	LOCAL CONST Robtarget Tr_meulage_bavure_P270 :=[[-219.63696875,-205.171546875,20],[0.53729501780428,-0.564922938891818,0.453775369108491,-0.431583191687283],[0,0,0,0],[8.999999E+09,8.999999E+09,8.999999E+09,8.999999E+09,8.999999E+09,8.999999E+09]];
	LOCAL CONST Robtarget Tr_meulage_bavure_P271 :=[[-219.324734375,-207.44634375,20],[0.537993238973984,-0.564758927457813,0.45310570554085,-0.431631611772482],[0,0,0,0],[8.999999E+09,8.999999E+09,8.999999E+09,8.999999E+09,8.999999E+09,8.999999E+09]];
	LOCAL CONST Robtarget Tr_meulage_bavure_P272 :=[[-219.077484375,-208.372515625,20],[0.538304707849301,-0.564135132378618,0.452955772497051,-0.432215990084863],[0,0,0,0],[8.999999E+09,8.999999E+09,8.999999E+09,8.999999E+09,8.999999E+09,8.999999E+09]];
	LOCAL CONST Robtarget Tr_meulage_bavure_P273 :=[[-218.728875,-210.97625,20],[0.538253392960368,-0.56310894895446,0.453282288328033,-0.433274466893857],[0,0,0,0],[8.999999E+09,8.999999E+09,8.999999E+09,8.999999E+09,8.999999E+09,8.999999E+09]];
	LOCAL CONST Robtarget Tr_meulage_bavure_P274 :=[[-218.566671875,-211.56171875,20],[0.537902797214692,-0.561749600415359,0.453996649502375,-0.434724061241626],[0,0,0,0],[8.999999E+09,8.999999E+09,8.999999E+09,8.999999E+09,8.999999E+09,8.999999E+09]];
	LOCAL CONST Robtarget Tr_meulage_bavure_P275 :=[[-217.610703125,-218.654484375,20],[0.537331594068803,-0.560152131881694,0.454988034586502,-0.436451870825392],[0,0,0,0],[8.999999E+09,8.999999E+09,8.999999E+09,8.999999E+09,8.999999E+09,8.999999E+09]];
	LOCAL CONST Robtarget Tr_meulage_bavure_P276 :=[[-217.24321875,-220.540375,20],[0.536643862605788,-0.558402103153409,0.456123837189228,-0.438350888067042],[0,0,0,0],[8.999999E+09,8.999999E+09,8.999999E+09,8.999999E+09,8.999999E+09,8.999999E+09]];
	LOCAL CONST Robtarget Tr_meulage_bavure_P277 :=[[-217.107078125,-221.269171875,20],[0.535921621847869,-0.55659175325912,0.457294923702402,-0.440312375701505],[0,0,0,0],[8.999999E+09,8.999999E+09,8.999999E+09,8.999999E+09,8.999999E+09,8.999999E+09]];
	LOCAL CONST Robtarget Tr_meulage_bavure_P278 :=[[-216.99709375,-221.83040625,20],[0.535229940524766,-0.55481109003148,0.458413067683216,-0.44223412862555],[0,0,0,0],[8.999999E+09,8.999999E+09,8.999999E+09,8.999999E+09,8.999999E+09,8.999999E+09]];
	LOCAL CONST Robtarget Tr_meulage_bavure_P279 :=[[-215.919453125,-225.61296875,20],[0.534637158213425,-0.553121918752511,0.459395983531932,-0.44404344648665],[0,0,0,0],[8.999999E+09,8.999999E+09,8.999999E+09,8.999999E+09,8.999999E+09,8.999999E+09]];
	LOCAL CONST Robtarget Tr_meulage_bavure_P280 :=[[-215.4938125,-227.822453125,20],[0.534190972566451,-0.551569737548126,0.460187785384334,-0.445688267326685],[0,0,0,0],[8.999999E+09,8.999999E+09,8.999999E+09,8.999999E+09,8.999999E+09,8.999999E+09]];
	LOCAL CONST Robtarget Tr_meulage_bavure_P281 :=[[-215.101453125,-230.017,20],[0.533919682326157,-0.550203109380352,0.460752711338939,-0.447116595807787],[0,0,0,0],[8.999999E+09,8.999999E+09,8.999999E+09,8.999999E+09,8.999999E+09,8.999999E+09]];
	LOCAL CONST Robtarget Tr_meulage_bavure_P282 :=[[-214.766375,-231.03446875,20],[0.533869793524164,-0.549045269612884,0.461042387233755,-0.448299289149539],[0,0,0,0],[8.999999E+09,8.999999E+09,8.999999E+09,8.999999E+09,8.999999E+09,8.999999E+09]];
	LOCAL CONST Robtarget Tr_meulage_bavure_P283 :=[[-214.39034375,-233.601546875,20],[0.534074564116095,-0.548144938680638,0.461016631292879,-0.449182759947851],[0,0,0,0],[8.999999E+09,8.999999E+09,8.999999E+09,8.999999E+09,8.999999E+09,8.999999E+09]];
	LOCAL CONST Robtarget Tr_meulage_bavure_P284 :=[[-214.230546875,-234.2085625,20],[0.534566009335567,-0.547535508259174,0.460639359023246,-0.449728173208069],[0,0,0,0],[8.999999E+09,8.999999E+09,8.999999E+09,8.999999E+09,8.999999E+09,8.999999E+09]];
	LOCAL CONST Robtarget Tr_meulage_bavure_P285 :=[[-213.2238125,-241.16003125,20],[0.535386335741234,-0.547259939100456,0.459861332170375,-0.449883969187421],[0,0,0,0],[8.999999E+09,8.999999E+09,8.999999E+09,8.999999E+09,8.999999E+09,8.999999E+09]];
	LOCAL CONST Robtarget Tr_meulage_bavure_P286 :=[[-212.793484375,-243.30528125,20],[0.536594038742582,-0.547390070776213,0.458609537333498,-0.449564500676256],[0,0,0,0],[8.999999E+09,8.999999E+09,8.999999E+09,8.999999E+09,8.999999E+09,8.999999E+09]];
	LOCAL CONST Robtarget Tr_meulage_bavure_P287 :=[[-212.653484375,-243.93984375,20],[0.538255330930929,-0.54797778261946,0.456804384011849,-0.448699569007427],[0,0,0,0],[8.999999E+09,8.999999E+09,8.999999E+09,8.999999E+09,8.999999E+09,8.999999E+09]];
	LOCAL CONST Robtarget Tr_meulage_bavure_P288 :=[[-212.53553125,-244.61078125,20],[0.540450412619775,-0.549105109829106,0.454341727655778,-0.447180639528864],[0,0,0,0],[8.999999E+09,8.999999E+09,8.999999E+09,8.999999E+09,8.999999E+09,8.999999E+09]];
	LOCAL CONST Robtarget Tr_meulage_bavure_P289 :=[[-211.432546875,-248.382609375,20],[0.543265483790806,-0.550855839481898,0.451104099741733,-0.44488824374941],[0,0,0,0],[8.999999E+09,8.999999E+09,8.999999E+09,8.999999E+09,8.999999E+09,8.999999E+09]];
	LOCAL CONST Robtarget Tr_meulage_bavure_P290 :=[[-210.87403125,-250.098296875,20],[0.546796245142534,-0.553313577146664,0.446954285400637,-0.441689730925675],[0,0,0,0],[8.999999E+09,8.999999E+09,8.999999E+09,8.999999E+09,8.999999E+09,8.999999E+09]];
	LOCAL CONST Robtarget Tr_meulage_bavure_P291 :=[[-210.5504375,-252.859703125,20],[0.551129613263795,-0.556588605739961,0.441743303392717,-0.43741070774712],[0,0,0,0],[8.999999E+09,8.999999E+09,8.999999E+09,8.999999E+09,8.999999E+09,8.999999E+09]];
	LOCAL CONST Robtarget Tr_meulage_bavure_P292 :=[[-210.326328125,-253.7085625,20],[0.556352636409364,-0.560749575377414,0.435311239016695,-0.431897884759985],[0,0,0,0],[8.999999E+09,8.999999E+09,8.999999E+09,8.999999E+09,8.999999E+09,8.999999E+09]];
	LOCAL CONST Robtarget Tr_meulage_bavure_P293 :=[[-209.778859375,-256.37915625,20],[0.562534887167558,-0.565860689136051,0.427491552289097,-0.424979004106455],[0,0,0,0],[8.999999E+09,8.999999E+09,8.999999E+09,8.999999E+09,8.999999E+09,8.999999E+09]];
	LOCAL CONST Robtarget Tr_meulage_bavure_P294 :=[[-209.6011875,-256.862328125,20],[0.569700795502199,-0.571957017682978,0.418140443553853,-0.416490987888025],[0,0,0,0],[8.999999E+09,8.999999E+09,8.999999E+09,8.999999E+09,8.999999E+09,8.999999E+09]];
	LOCAL CONST Robtarget Tr_meulage_bavure_P295 :=[[-208.96625,-259.827125,20],[0.577848420825114,-0.579022623980751,0.407121335426489,-0.406295731836946],[0,0,0,0],[8.999999E+09,8.999999E+09,8.999999E+09,8.999999E+09,8.999999E+09,8.999999E+09]];
	LOCAL CONST Robtarget Tr_meulage_bavure_P296 :=[[-208.80403125,-260.40115625,20],[0.586930696044148,-0.586995327394604,0.394324157697137,-0.394280740481293],[0,0,0,0],[8.999999E+09,8.999999E+09,8.999999E+09,8.999999E+09,8.999999E+09,8.999999E+09]];
	LOCAL CONST Robtarget Tr_meulage_bavure_P297 :=[[-206.9465625,-264.3128125,20],[0.596830556528174,-0.595758661219479,0.379700963340443,-0.380384125345135],[0,0,0,0],[8.999999E+09,8.999999E+09,8.999999E+09,8.999999E+09,8.999999E+09,8.999999E+09]];
	LOCAL CONST Robtarget Tr_meulage_bavure_P298 :=[[-204.21284375,-269.3765625,20],[0.607373754979424,-0.60515091678245,0.363261810220388,-0.364596142210751],[0,0,0,0],[8.999999E+09,8.999999E+09,8.999999E+09,8.999999E+09,8.999999E+09,8.999999E+09]];
	LOCAL CONST Robtarget Tr_meulage_bavure_P299 :=[[-204.11028125,-269.53403125,20],[0.618359765363299,-0.61496081647422,0.345061273014783,-0.346968460593501],[0,0,0,0],[8.999999E+09,8.999999E+09,8.999999E+09,8.999999E+09,8.999999E+09,8.999999E+09]];
	LOCAL CONST Robtarget Tr_meulage_bavure_P300 :=[[-203.988234375,-269.722875,20],[0.629554145495922,-0.624946065590333,0.325221808959532,-0.327619852831222],[0,0,0,0],[8.999999E+09,8.999999E+09,8.999999E+09,8.999999E+09,8.999999E+09,8.999999E+09]];
	LOCAL CONST Robtarget Tr_meulage_bavure_P301 :=[[-202.10503125,-271.81009375,20],[0.640691980291868,-0.634846776112635,0.303952512068475,-0.306751084197502],[0,0,0,0],[8.999999E+09,8.999999E+09,8.999999E+09,8.999999E+09,8.999999E+09,8.999999E+09]];
	LOCAL CONST Robtarget Tr_meulage_bavure_P302 :=[[-198.574953125,-275.987625,20],[0.651514894985457,-0.64441431008127,0.28151592453752,-0.284617853983822],[0,0,0,0],[8.999999E+09,8.999999E+09,8.999999E+09,8.999999E+09,8.999999E+09,8.999999E+09]];
	LOCAL CONST Robtarget Tr_meulage_bavure_P303 :=[[-198.1525625,-276.32359375,20],[0.661778551172858,-0.653403298900412,0.258256180431549,-0.261566480005598],[0,0,0,0],[8.999999E+09,8.999999E+09,8.999999E+09,8.999999E+09,8.999999E+09,8.999999E+09]];
	LOCAL CONST Robtarget Tr_meulage_bavure_P304 :=[[-198.02296875,-276.43640625,20],[0.671270334947485,-0.661609679683465,0.234574203209948,-0.237999395707325],[0,0,0,0],[8.999999E+09,8.999999E+09,8.999999E+09,8.999999E+09,8.999999E+09,8.999999E+09]];
	LOCAL CONST Robtarget Tr_meulage_bavure_P305 :=[[-193.361921875,-279.8115,20],[0.679821587865466,-0.668886501373737,0.210911256713211,-0.214359274918843],[0,0,0,0],[8.999999E+09,8.999999E+09,8.999999E+09,8.999999E+09,8.999999E+09,8.999999E+09]];
	LOCAL CONST Robtarget Tr_meulage_bavure_P306 :=[[-192.662015625,-280.25846875,20],[0.687332808397279,-0.675135741510664,0.187723907861307,-0.191115345937563],[0,0,0,0],[8.999999E+09,8.999999E+09,8.999999E+09,8.999999E+09,8.999999E+09,8.999999E+09]];
	LOCAL CONST Robtarget Tr_meulage_bavure_P307 :=[[-185.646046875,-284.1375,20],[0.693782149187908,-0.680318577808721,0.165437229325596,-0.168711248319718],[0,0,0,0],[8.999999E+09,8.999999E+09,8.999999E+09,8.999999E+09,8.999999E+09,8.999999E+09]];
	LOCAL CONST Robtarget Tr_meulage_bavure_P308 :=[[-185.354671875,-284.25996875,20],[0.699188719439392,-0.684470610463102,0.144444095505406,-0.147550063688893],[0,0,0,0],[8.999999E+09,8.999999E+09,8.999999E+09,8.999999E+09,8.999999E+09,8.999999E+09]];
	LOCAL CONST Robtarget Tr_meulage_bavure_P309 :=[[-180.695234375,-286.03475,20],[0.70362823463154,-0.687682408745583,0.125033593354582,-0.127932844352095],[0,0,0,0],[8.999999E+09,8.999999E+09,8.999999E+09,8.999999E+09,8.999999E+09,8.999999E+09]];
	LOCAL CONST Robtarget Tr_meulage_bavure_P310 :=[[-179.823375,-286.31721875,20],[0.707229971052489,-0.690061561664037,0.107377724376658,-0.110049232012663],[0,0,0,0],[8.999999E+09,8.999999E+09,8.999999E+09,8.999999E+09,8.999999E+09,8.999999E+09]];
	LOCAL CONST Robtarget Tr_meulage_bavure_P311 :=[[-179.685515625,-286.362125,20],[0.71011625284017,-0.691753966347935,0.0915438463828495,-0.0939738351008869],[0,0,0,0],[8.999999E+09,8.999999E+09,8.999999E+09,8.999999E+09,8.999999E+09,8.999999E+09]];
	LOCAL CONST Robtarget Tr_meulage_bavure_P312 :=[[-179.47846875,-286.4050625,20],[0.712422501657508,-0.692893522682186,0.0774902952212525,-0.0796743340333189],[0,0,0,0],[8.999999E+09,8.999999E+09,8.999999E+09,8.999999E+09,8.999999E+09,8.999999E+09]];
	LOCAL CONST Robtarget Tr_meulage_bavure_P313 :=[[-176.450546875,-286.82434375,20],[0.714278213115217,-0.693598764499872,0.0650809529079148,-0.0670213228889187],[0,0,0,0],[8.999999E+09,8.999999E+09,8.999999E+09,8.999999E+09,8.999999E+09,8.999999E+09]];
	LOCAL CONST Robtarget Tr_meulage_bavure_P314 :=[[-174.725015625,-287.0270625,20],[0.715791157369704,-0.693969981495662,0.0541362999646006,-0.0558385605150519],[0,0,0,0],[8.999999E+09,8.999999E+09,8.999999E+09,8.999999E+09,8.999999E+09,8.999999E+09]];
	LOCAL CONST Robtarget Tr_meulage_bavure_P315 :=[[-172.48009375,-287.12125,20],[0.717041268538116,-0.694095069222552,0.0444470233568255,-0.045916404572963],[0,0,0,0],[8.999999E+09,8.999999E+09,8.999999E+09,8.999999E+09,8.999999E+09,8.999999E+09]];
	LOCAL CONST Robtarget Tr_meulage_bavure_P316 :=[[-170.3138125,-287.373625,20],[0.718086151112885,-0.694044263785635,0.0358082882651692,-0.0370486973813791],[0,0,0,0],[8.999999E+09,8.999999E+09,8.999999E+09,8.999999E+09,8.999999E+09,8.999999E+09]];
	LOCAL CONST Robtarget Tr_meulage_bavure_P317 :=[[-169.579875,-287.35590625,20],[0.718985888631994,-0.693850501788261,0.0280425230376692,-0.0290583898026416],[0,0,0,0],[8.999999E+09,8.999999E+09,8.999999E+09,8.999999E+09,8.999999E+09,8.999999E+09]];
	LOCAL CONST Robtarget Tr_meulage_bavure_P318 :=[[-166.023984375,-287.1190625,20],[0.719774919648292,-0.693547646838508,0.0209970440043696,-0.0217910704909592],[0,0,0,0],[8.999999E+09,8.999999E+09,8.999999E+09,8.999999E+09,8.999999E+09,8.999999E+09]];
	LOCAL CONST Robtarget Tr_meulage_bavure_P319 :=[[-160.928265625,-287.3099375,20],[0.720464951309386,-0.693172347648877,0.0145821147957829,-0.0151562633188785],[0,0,0,0],[8.999999E+09,8.999999E+09,8.999999E+09,8.999999E+09,8.999999E+09,8.999999E+09]];
	LOCAL CONST Robtarget Tr_meulage_bavure_P320 :=[[-160.79965625,-287.30678125,20],[0.721085760434946,-0.692731207117006,0.00873022747837951,-0.00908756911099294],[0,0,0,0],[8.999999E+09,8.999999E+09,8.999999E+09,8.999999E+09,8.999999E+09,8.999999E+09]];
	LOCAL CONST Robtarget Tr_meulage_bavure_P321 :=[[-158.17290625,-287.03840625,20],[0.721652690962883,-0.692237672883823,0.00341929407178484,-0.00356458896236797],[0,0,0,0],[8.999999E+09,8.999999E+09,8.999999E+09,8.999999E+09,8.999999E+09,8.999999E+09]];
	LOCAL CONST Robtarget Tr_meulage_bavure_P322 :=[[-156.189484375,-287.00271875,20],[0.722168553326168,-0.691714363171503,-0.00135201117505688,0.00141153633111643],[0,0,0,0],[8.999999E+09,8.999999E+09,8.999999E+09,8.999999E+09,8.999999E+09,8.999999E+09]];
	LOCAL CONST Robtarget Tr_meulage_bavure_P323 :=[[-152.667203125,-287.19778125,20],[0.722648884556597,-0.691168089401874,-0.00558376990281725,0.00583809518084595],[0,0,0,0],[8.999999E+09,8.999999E+09,8.999999E+09,8.999999E+09,8.999999E+09,8.999999E+09]];
	LOCAL CONST Robtarget Tr_meulage_bavure_P324 :=[[-149.589046875,-287.21059375,20],[0.723113666831497,-0.690599316019845,-0.00924582442862393,0.00968113036079282],[0,0,0,0],[8.999999E+09,8.999999E+09,8.999999E+09,8.999999E+09,8.999999E+09,8.999999E+09]];
	LOCAL CONST Robtarget Tr_meulage_bavure_P325 :=[[-144.85625,-286.99990625,20],[0.72355718246237,-0.690033503818427,-0.0123218608697659,0.0129204899244532],[0,0,0,0],[8.999999E+09,8.999999E+09,8.999999E+09,8.999999E+09,8.999999E+09,8.999999E+09]];
	LOCAL CONST Robtarget Tr_meulage_bavure_P326 :=[[-143.57653125,-287.2320625,20],[0.723999358467151,-0.689466631061457,-0.0148019658892337,0.0155433393366104],[0,0,0,0],[8.999999E+09,8.999999E+09,8.999999E+09,8.999999E+09,8.999999E+09,8.999999E+09]];
	LOCAL CONST Robtarget Tr_meulage_bavure_P327 :=[[-140.72509375,-287.0025,20],[0.724444298776135,-0.688908293410537,-0.0166790464051948,0.0175394028390153],[0,0,0,0],[8.999999E+09,8.999999E+09,8.999999E+09,8.999999E+09,8.999999E+09,8.999999E+09]];
	LOCAL CONST Robtarget Tr_meulage_bavure_P328 :=[[-139.5401875,-286.91978125,20],[0.72490078853614,-0.688359587713625,-0.0179553342944921,0.0189084836193525],[0,0,0,0],[8.999999E+09,8.999999E+09,8.999999E+09,8.999999E+09,8.999999E+09,8.999999E+09]];
	LOCAL CONST Robtarget Tr_meulage_bavure_P329 :=[[-137.21515625,-287.07465625,20],[0.725359692131602,-0.687835653160883,-0.0186601652392554,0.0196781478989506],[0,0,0,0],[8.999999E+09,8.999999E+09,8.999999E+09,8.999999E+09,8.999999E+09,8.999999E+09]];
	LOCAL CONST Robtarget Tr_meulage_bavure_P330 :=[[-135.483828125,-287.07825,20],[0.725833732047821,-0.687323758836874,-0.0188483306036036,0.0199043812599118],[0,0,0,0],[8.999999E+09,8.999999E+09,8.999999E+09,8.999999E+09,8.999999E+09,8.999999E+09]];
	LOCAL CONST Robtarget Tr_meulage_bavure_P331 :=[[-132.387421875,-286.80325,20],[0.726321044579261,-0.686822734580372,-0.018592585476214,0.0196618216383935],[0,0,0,0],[8.999999E+09,8.999999E+09,8.999999E+09,8.999999E+09,8.999999E+09,8.999999E+09]];
	LOCAL CONST Robtarget Tr_meulage_bavure_P332 :=[[-130.4786953125,-286.93715625,20],[0.726812176110579,-0.68633672027097,-0.0179819950748647,0.0190424504258088],[0,0,0,0],[8.999999E+09,8.999999E+09,8.999999E+09,8.999999E+09,8.999999E+09,8.999999E+09]];
	LOCAL CONST Robtarget Tr_meulage_bavure_P333 :=[[-129.3878515625,-286.88765625,20],[0.727297328990863,-0.685868930510056,-0.0171164226950637,0.0181503024181905],[0,0,0,0],[8.999999E+09,8.999999E+09,8.999999E+09,8.999999E+09,8.999999E+09,8.999999E+09]];
	LOCAL CONST Robtarget Tr_meulage_bavure_P334 :=[[-126.4455859375,-287.0436875,20],[0.727787757509097,-0.68540016068255,-0.0161018599931864,0.0170976565930428],[0,0,0,0],[8.999999E+09,8.999999E+09,8.999999E+09,8.999999E+09,8.999999E+09,8.999999E+09]];
	LOCAL CONST Robtarget Tr_meulage_bavure_P335 :=[[-126.3676171875,-287.04559375,20],[0.72827628013861,-0.684932120707197,-0.0150354989508349,0.0159869816510227],[0,0,0,0],[8.999999E+09,8.999999E+09,8.999999E+09,8.999999E+09,8.999999E+09,8.999999E+09]];
	LOCAL CONST Robtarget Tr_meulage_bavure_P336 :=[[-122.262265625,-286.86140625,20],[0.728755053664664,-0.684469256132264,-0.0139954111703684,0.0149009272909549],[0,0,0,0],[8.999999E+09,8.999999E+09,8.999999E+09,8.999999E+09,8.999999E+09,8.999999E+09]];
	LOCAL CONST Robtarget Tr_meulage_bavure_P337 :=[[-120.081265625,-287.044,20],[0.729234909118417,-0.683998119330656,-0.0130346409279294,0.0138966978473149],[0,0,0,0],[8.999999E+09,8.999999E+09,8.999999E+09,8.999999E+09,8.999999E+09,8.999999E+09]];
	LOCAL CONST Robtarget Tr_meulage_bavure_P338 :=[[-118.7465546875,-287.03021875,20],[0.729708993844251,-0.683525414703059,-0.0121869491838472,0.013010381524496],[0,0,0,0],[8.999999E+09,8.999999E+09,8.999999E+09,8.999999E+09,8.999999E+09,8.999999E+09]];
	LOCAL CONST Robtarget Tr_meulage_bavure_P339 :=[[-116.7078515625,-287.04834375,20],[0.730167601402134,-0.683061652581515,-0.011473244296343,0.0122644731064913],[0,0,0,0],[8.999999E+09,8.999999E+09,8.999999E+09,8.999999E+09,8.999999E+09,8.999999E+09]];
	LOCAL CONST Robtarget Tr_meulage_bavure_P340 :=[[-116.34390625,-287.02965625,20],[0.730618690391253,-0.682598813248682,-0.0109056678682374,0.0116728664349885],[0,0,0,0],[8.999999E+09,8.999999E+09,8.999999E+09,8.999999E+09,8.999999E+09,8.999999E+09]];
	LOCAL CONST Robtarget Tr_meulage_bavure_P341 :=[[-115.980984375,-287.02528125,20],[0.731069622640329,-0.682129611176638,-0.0104891996973489,0.0112417569020533],[0,0,0,0],[8.999999E+09,8.999999E+09,8.999999E+09,8.999999E+09,8.999999E+09,8.999999E+09]];
	LOCAL CONST Robtarget Tr_meulage_bavure_P342 :=[[-110.514953125,-286.68334375,20],[0.731512446344771,-0.681663052915111,-0.0102266220917813,0.0109744855793644],[0,0,0,0],[8.999999E+09,8.999999E+09,8.999999E+09,8.999999E+09,8.999999E+09,8.999999E+09]];
	LOCAL CONST Robtarget Tr_meulage_bavure_P343 :=[[-109.358828125,-286.5719375,20],[0.731948684007435,-0.681197789056066,-0.010120886435774,0.0108749171337133],[0,0,0,0],[8.999999E+09,8.999999E+09,8.999999E+09,8.999999E+09,8.999999E+09,8.999999E+09]];
	LOCAL CONST Robtarget Tr_meulage_bavure_P344 :=[[-106.400546875,-286.3830625,20],[0.732377372221076,-0.680735183537822,-0.0101665535442954,0.0109378124553808],[0,0,0,0],[8.999999E+09,8.999999E+09,8.999999E+09,8.999999E+09,8.999999E+09,8.999999E+09]];
	LOCAL CONST Robtarget Tr_meulage_bavure_P345 :=[[-101.39840625,-286.41196875,20],[0.732805623556927,-0.68026822878917,-0.0103416071680586,0.0111402937380435],[0,0,0,0],[8.999999E+09,8.999999E+09,8.999999E+09,8.999999E+09,8.999999E+09,8.999999E+09]];
	LOCAL CONST Robtarget Tr_meulage_bavure_P346 :=[[-97.4696328125,-286.269125,20],[0.733233045106648,-0.679798118853771,-0.0106161447322498,0.0114506173427568],[0,0,0,0],[8.999999E+09,8.999999E+09,8.999999E+09,8.999999E+09,8.999999E+09,8.999999E+09]];
	LOCAL CONST Robtarget Tr_meulage_bavure_P347 :=[[-92.7008046875,-286.2609375,20],[0.733644287088494,-0.679342872996497,-0.010941179119575,0.0118157323409935],[0,0,0,0],[8.999999E+09,8.999999E+09,8.999999E+09,8.999999E+09,8.999999E+09,8.999999E+09]];
	LOCAL CONST Robtarget Tr_meulage_bavure_P348 :=[[-87.303921875,-286.25903125,20],[0.734060236148746,-0.678881747816684,-0.0112624397148181,0.0121778338911871],[0,0,0,0],[8.999999E+09,8.999999E+09,8.999999E+09,8.999999E+09,8.999999E+09,8.999999E+09]];
	LOCAL CONST Robtarget Tr_meulage_bavure_P349 :=[[-85.25515625,-286.0718125,20],[0.734471125173337,-0.678427045037026,-0.0115331468776594,0.0124858869144309],[0,0,0,0],[8.999999E+09,8.999999E+09,8.999999E+09,8.999999E+09,8.999999E+09,8.999999E+09]];
	LOCAL CONST Robtarget Tr_meulage_bavure_P350 :=[[-80.46753125,-286.2709375,20],[0.734882405250611,-0.677974573350089,-0.0117118487695932,0.0126949179689748],[0,0,0,0],[8.999999E+09,8.999999E+09,8.999999E+09,8.999999E+09,8.999999E+09,8.999999E+09]];
	LOCAL CONST Robtarget Tr_meulage_bavure_P351 :=[[-75.5986953125,-286.21459375,20],[0.735294200384523,-0.677524835745839,-0.0117863499460959,0.0127913167190786],[0,0,0,0],[8.999999E+09,8.999999E+09,8.999999E+09,8.999999E+09,8.999999E+09,8.999999E+09]];
	LOCAL CONST Robtarget Tr_meulage_bavure_P352 :=[[-72.818390625,-286.01653125,20],[0.735702295195481,-0.677082212616164,-0.0117645118239197,0.0127830537997292],[0,0,0,0],[8.999999E+09,8.999999E+09,8.999999E+09,8.999999E+09,8.999999E+09,8.999999E+09]];
	LOCAL CONST Robtarget Tr_meulage_bavure_P353 :=[[-70.6874375,-286.05234375,20],[0.73610404458772,-0.676648080873107,-0.0116866183362495,0.0127135024365487],[0,0,0,0],[8.999999E+09,8.999999E+09,8.999999E+09,8.999999E+09,8.999999E+09,8.999999E+09]];
	LOCAL CONST Robtarget Tr_meulage_bavure_P354 :=[[-68.363375,-286.02184375,20],[0.736508513607693,-0.676210358433826,-0.0116112907362422,0.0126466777306154],[0,0,0,0],[8.999999E+09,8.999999E+09,8.999999E+09,8.999999E+09,8.999999E+09,8.999999E+09]];
	LOCAL CONST Robtarget Tr_meulage_bavure_P355 :=[[-67.0465703125,-285.9046875,20],[0.736905504555383,-0.67577833986711,-0.0115871676885302,0.0126352786825977],[0,0,0,0],[8.999999E+09,8.999999E+09,8.999999E+09,8.999999E+09,8.999999E+09,8.999999E+09]];
	LOCAL CONST Robtarget Tr_meulage_bavure_P356 :=[[-63.81491015625,-286.06209375,20],[0.737301936439538,-0.675342882527419,-0.0116569401123361,0.0127264012698559],[0,0,0,0],[8.999999E+09,8.999999E+09,8.999999E+09,8.999999E+09,8.999999E+09,8.999999E+09]];
	LOCAL CONST Robtarget Tr_meulage_bavure_P357 :=[[-61.29443359375,-286.0691875,20],[0.737695697156239,-0.674905224600262,-0.0118462900863419,0.0129484213566949],[0,0,0,0],[8.999999E+09,8.999999E+09,8.999999E+09,8.999999E+09,8.999999E+09,8.999999E+09]];
	LOCAL CONST Robtarget Tr_meulage_bavure_P358 :=[[-59.2204296875,-286.01996875,20],[0.73807842663314,-0.674474572683839,-0.0121478869477723,0.0132934489281806],[0,0,0,0],[8.999999E+09,8.999999E+09,8.999999E+09,8.999999E+09,8.999999E+09,8.999999E+09]];
	LOCAL CONST Robtarget Tr_meulage_bavure_P359 :=[[-57.1460859375,-285.81696875,20],[0.738457651594908,-0.674043842272608,-0.0125255174570652,0.0137224964108707],[0,0,0,0],[8.999999E+09,8.999999E+09,8.999999E+09,8.999999E+09,8.999999E+09,8.999999E+09]];
	LOCAL CONST Robtarget Tr_meulage_bavure_P360 :=[[-52.2008359375,-285.65203125,20],[0.738836754060016,-0.673611280001105,-0.0129261397147576,0.0141777719478838],[0,0,0,0],[8.999999E+09,8.999999E+09,8.999999E+09,8.999999E+09,8.999999E+09,8.999999E+09]];
	LOCAL CONST Robtarget Tr_meulage_bavure_P361 :=[[-50.8576953125,-285.7155625,20],[0.739216919954698,-0.673178446098049,-0.0132818711139443,0.0145848161256416],[0,0,0,0],[8.999999E+09,8.999999E+09,8.999999E+09,8.999999E+09,8.999999E+09,8.999999E+09]];
	LOCAL CONST Robtarget Tr_meulage_bavure_P362 :=[[-48.06460546875,-285.51146875,20],[0.739594408421707,-0.672752103413518,-0.0135369065780215,0.0148818864506438],[0,0,0,0],[8.999999E+09,8.999999E+09,8.999999E+09,8.999999E+09,8.999999E+09,8.999999E+09]];
	LOCAL CONST Robtarget Tr_meulage_bavure_P363 :=[[-46.638671875,-285.55459375,20],[0.73996808302208,-0.672335946508094,-0.0136432956714231,0.0150157126009993],[0,0,0,0],[8.999999E+09,8.999999E+09,8.999999E+09,8.999999E+09,8.999999E+09,8.999999E+09]];
	LOCAL CONST Robtarget Tr_meulage_bavure_P364 :=[[-44.5212421875,-285.5055,20],[0.740350610592449,-0.671917428103571,-0.0135738910831586,0.0149563594144233],[0,0,0,0],[8.999999E+09,8.999999E+09,8.999999E+09,8.999999E+09,8.999999E+09,8.999999E+09]];
	LOCAL CONST Robtarget Tr_meulage_bavure_P365 :=[[-42.613890625,-285.28371875,20],[0.740729955907969,-0.671509509518791,-0.0133335891229953,0.0147080402334867],[0,0,0,0],[8.999999E+09,8.999999E+09,8.999999E+09,8.999999E+09,8.999999E+09,8.999999E+09]];
	LOCAL CONST Robtarget Tr_meulage_bavure_P366 :=[[-39.94320703125,-285.19134375,20],[0.741104920372723,-0.671112719565838,-0.0129326831912417,0.0142814684735096],[0,0,0,0],[8.999999E+09,8.999999E+09,8.999999E+09,8.999999E+09,8.999999E+09,8.999999E+09]];
	LOCAL CONST Robtarget Tr_meulage_bavure_P367 :=[[-39.05349609375,-285.2751875,20],[0.741486808866516,-0.670711839125037,-0.0124228214703777,0.0137337045685749],[0,0,0,0],[8.999999E+09,8.999999E+09,8.999999E+09,8.999999E+09,8.999999E+09,8.999999E+09]];
	LOCAL CONST Robtarget Tr_meulage_bavure_P368 :=[[-36.61151171875,-285.167125,20],[0.741875276336261,-0.670304094514672,-0.0118701288053807,0.0131375522836614],[0,0,0,0],[8.999999E+09,8.999999E+09,8.999999E+09,8.999999E+09,8.999999E+09,8.999999E+09]];
	LOCAL CONST Robtarget Tr_meulage_bavure_P369 :=[[-34.20391796875,-284.9718125,20],[0.742258408201348,-0.669900950100451,-0.011314265228886,0.0125363436154277],[0,0,0,0],[8.999999E+09,8.999999E+09,8.999999E+09,8.999999E+09,8.999999E+09,8.999999E+09]];
	LOCAL CONST Robtarget Tr_meulage_bavure_P370 :=[[-32.377166015625,-285.07184375,20],[0.7426351259316,-0.669502100752265,-0.0107969423318776,0.0119763457340922],[0,0,0,0],[8.999999E+09,8.999999E+09,8.999999E+09,8.999999E+09,8.999999E+09,8.999999E+09]];
	LOCAL CONST Robtarget Tr_meulage_bavure_P371 :=[[-29.942443359375,-285.0098125,20],[0.743018422986564,-0.669092438878601,-0.0103436679200184,0.0114865082599196],[0,0,0,0],[8.999999E+09,8.999999E+09,8.999999E+09,8.999999E+09,8.999999E+09,8.999999E+09]];
	LOCAL CONST Robtarget Tr_meulage_bavure_P372 :=[[-28.338623046875,-285.10840625,20],[0.743397237835754,-0.66868442589708,-0.00995721397532873,0.0110697439317037],[0,0,0,0],[8.999999E+09,8.999999E+09,8.999999E+09,8.999999E+09,8.999999E+09,8.999999E+09]];
	LOCAL CONST Robtarget Tr_meulage_bavure_P373 :=[[-26.397857421875,-285.09925,20],[0.74377973357237,-0.66827024988322,-0.00960599218357905,0.0106913966441709],[0,0,0,0],[8.999999E+09,8.999999E+09,8.999999E+09,8.999999E+09,8.999999E+09,8.999999E+09]];
	LOCAL CONST Robtarget Tr_meulage_bavure_P374 :=[[-24.54379296875,-284.91765625,20],[0.744160644212133,-0.667858097670734,-0.00921869857605938,0.0102719315601381],[0,0,0,0],[8.999999E+09,8.999999E+09,8.999999E+09,8.999999E+09,8.999999E+09,8.999999E+09]];
	LOCAL CONST Robtarget Tr_meulage_bavure_P375 :=[[-23.49786328125,-285.05778125,20],[0.744546099294175,-0.667443388325873,-0.00871412352322955,0.00972077451281972],[0,0,0,0],[8.999999E+09,8.999999E+09,8.999999E+09,8.999999E+09,8.999999E+09,8.999999E+09]];
	LOCAL CONST Robtarget Tr_meulage_bavure_P376 :=[[-21.1500859375,-285.0423125,20],[0.744921204100422,-0.667045240463476,-0.00797857833854392,0.00891005860236419],[0,0,0,0],[8.999999E+09,8.999999E+09,8.999999E+09,8.999999E+09,8.999999E+09,8.999999E+09]];
	LOCAL CONST Robtarget Tr_meulage_bavure_P377 :=[[-18.6988515625,-285.003875,20],[0.745306039021724,-0.666641983739337,-0.00690820100662859,0.00772337184666341],[0,0,0,0],[8.999999E+09,8.999999E+09,8.999999E+09,8.999999E+09,8.999999E+09,8.999999E+09]];
	LOCAL CONST Robtarget Tr_meulage_bavure_P378 :=[[-16.727111328125,-284.85565625,20],[0.745698651308556,-0.66623340492249,-0.00543607405853542,0.00608446388895029],[0,0,0,0],[8.999999E+09,8.999999E+09,8.999999E+09,8.999999E+09,8.999999E+09,8.999999E+09]];
	LOCAL CONST Robtarget Tr_meulage_bavure_P379 :=[[-11.87109375,-285.08015625,20],[0.74610016280311,-0.665812895231184,-0.00350652612098457,0.00392936172981681],[0,0,0,0],[8.999999E+09,8.999999E+09,8.999999E+09,8.999999E+09,8.999999E+09,8.999999E+09]];
	LOCAL CONST Robtarget Tr_meulage_bavure_P380 :=[[-8.3177490234375,-285.1109375,20],[0.746496290504789,-0.665387334140756,-0.00114937578840505,0.0012894816573994],[0,0,0,0],[8.999999E+09,8.999999E+09,8.999999E+09,8.999999E+09,8.999999E+09,8.999999E+09]];
	LOCAL CONST Robtarget Tr_meulage_bavure_P381 :=[[-5.799560546875,-285.05053125,20],[0.746875495857413,-0.66496000565985,0.0015140932677863,-0.00170061229326133],[0,0,0,0],[8.999999E+09,8.999999E+09,8.999999E+09,8.999999E+09,8.999999E+09,8.999999E+09]];
	LOCAL CONST Robtarget Tr_meulage_bavure_P382 :=[[-3.87139892578125,-284.9315,20],[0.747250674864053,-0.664510321088494,0.00433023627871674,-0.00486940816252721],[0,0,0,0],[8.999999E+09,8.999999E+09,8.999999E+09,8.999999E+09,8.999999E+09,8.999999E+09]];
	LOCAL CONST Robtarget Tr_meulage_bavure_P383 :=[[-2.29058837890625,-284.71034375,20],[0.747611357979807,-0.664050746803346,0.00708626644239052,-0.0079779644906735],[0,0,0,0],[8.999999E+09,8.999999E+09,8.999999E+09,8.999999E+09,8.999999E+09,8.999999E+09]];
	LOCAL CONST Robtarget Tr_meulage_bavure_P384 :=[[-0.498443603515625,-284.361375,20],[0.74797342502485,-0.663573075497054,0.00953726955906979,-0.0107503219176564],[0,0,0,0],[8.999999E+09,8.999999E+09,8.999999E+09,8.999999E+09,8.999999E+09,8.999999E+09]];
	LOCAL CONST Robtarget Tr_meulage_bavure_P385 :=[[131.446953125,-282.32440625,20],[0.748338803865792,-0.663091402371405,0.011464312535184,-0.012938170965634],[0,0,0,0],[8.999999E+09,8.999999E+09,8.999999E+09,8.999999E+09,8.999999E+09,8.999999E+09]];
	LOCAL CONST Robtarget Tr_meulage_bavure_P386 :=[[133.308234375,-282.79625,20],[0.748710944824383,-0.662620154013309,0.0126868303044676,-0.0143351641910574],[0,0,0,0],[8.999999E+09,8.999999E+09,8.999999E+09,8.999999E+09,8.999999E+09,8.999999E+09]];
	LOCAL CONST Robtarget Tr_meulage_bavure_P387 :=[[136.003296875,-282.894375,20],[0.749110427411547,-0.662149210130359,0.0131123063352003,-0.0148343685272678],[0,0,0,0],[8.999999E+09,8.999999E+09,8.999999E+09,8.999999E+09,8.999999E+09,8.999999E+09]];
	LOCAL CONST Robtarget Tr_meulage_bavure_P388 :=[[137.125359375,-282.668,20],[0.749524816555507,-0.661697206649568,0.0127192688351801,-0.0144075077612612],[0,0,0,0],[8.999999E+09,8.999999E+09,8.999999E+09,8.999999E+09,8.999999E+09,8.999999E+09]];
	LOCAL CONST Robtarget Tr_meulage_bavure_P389 :=[[138.402828125,-282.77528125,20],[0.749957697988967,-0.661254852884967,0.0115589940326936,-0.0131095545356023],[0,0,0,0],[8.999999E+09,8.999999E+09,8.999999E+09,8.999999E+09,8.999999E+09,8.999999E+09]];
	LOCAL CONST Robtarget Tr_meulage_bavure_P390 :=[[145.1876875,-282.74875,20],[0.750404048776996,-0.660815138530525,0.0097380795413633,-0.0110583034332436],[0,0,0,0],[8.999999E+09,8.999999E+09,8.999999E+09,8.999999E+09,8.999999E+09,8.999999E+09]];
	LOCAL CONST Robtarget Tr_meulage_bavure_P391 :=[[146.662296875,-282.71884375,20],[0.750858645720035,-0.660369545922452,0.00733492477328736,-0.00834001464140146],[0,0,0,0],[8.999999E+09,8.999999E+09,8.999999E+09,8.999999E+09,8.999999E+09,8.999999E+09]];
	LOCAL CONST Robtarget Tr_meulage_bavure_P392 :=[[147.953734375,-282.6699375,20],[0.751306586108964,-0.659919531807166,0.00440849957299088,-0.00501899792990888],[0,0,0,0],[8.999999E+09,8.999999E+09,8.999999E+09,8.999999E+09,8.999999E+09,8.999999E+09]];
	LOCAL CONST Robtarget Tr_meulage_bavure_P393 :=[[152.621453125,-282.3783125,20],[0.751747486400433,-0.659449376968218,0.000986072397507752,-0.0011240854448044],[0,0,0,0],[8.999999E+09,8.999999E+09,8.999999E+09,8.999999E+09,8.999999E+09,8.999999E+09]];
	LOCAL CONST Robtarget Tr_meulage_bavure_P394 :=[[153.813171875,-282.22275,20],[0.752158959088751,-0.658966153766303,-0.00298424182374386,0.00340628150776365],[0,0,0,0],[8.999999E+09,8.999999E+09,8.999999E+09,8.999999E+09,8.999999E+09,8.999999E+09]];
	LOCAL CONST Robtarget Tr_meulage_bavure_P395 :=[[156.108765625,-282.04996875,20],[0.752539307122924,-0.658445279346562,-0.00763408761414,0.00872502421060999],[0,0,0,0],[8.999999E+09,8.999999E+09,8.999999E+09,8.999999E+09,8.999999E+09,8.999999E+09]];
	LOCAL CONST Robtarget Tr_meulage_bavure_P396 :=[[157.16046875,-282.14321875,20],[0.752861812874993,-0.657876203597649,-0.0131270606302564,0.0150223744372718],[0,0,0,0],[8.999999E+09,8.999999E+09,8.999999E+09,8.999999E+09,8.999999E+09,8.999999E+09]];
	LOCAL CONST Robtarget Tr_meulage_bavure_P397 :=[[161.125359375,-282.1855625,20],[0.753094483874573,-0.657232769493895,-0.019657574244735,0.0225247605067908],[0,0,0,0],[8.999999E+09,8.999999E+09,8.999999E+09,8.999999E+09,8.999999E+09,8.999999E+09]];
	LOCAL CONST Robtarget Tr_meulage_bavure_P398 :=[[161.6613125,-282.136875,20],[0.753199280410119,-0.656466530884223,-0.0274272593114164,0.0314687665023153],[0,0,0,0],[8.999999E+09,8.999999E+09,8.999999E+09,8.999999E+09,8.999999E+09,8.999999E+09]];
	LOCAL CONST Robtarget Tr_meulage_bavure_P399 :=[[162.55315625,-282.20653125,20],[0.753104155367442,-0.655534205265269,-0.0366087134127631,0.0420575676636907],[0,0,0,0],[8.999999E+09,8.999999E+09,8.999999E+09,8.999999E+09,8.999999E+09,8.999999E+09]];
	LOCAL CONST Robtarget Tr_meulage_bavure_P400 :=[[164.935125,-282.16965625,20],[0.752729106259223,-0.654365515474713,-0.0473314614476047,0.054446280910069],[0,0,0,0],[8.999999E+09,8.999999E+09,8.999999E+09,8.999999E+09,8.999999E+09,8.999999E+09]];
	LOCAL CONST Robtarget Tr_meulage_bavure_P401 :=[[167.379390625,-281.97934375,20],[0.751970230020248,-0.65288729983475,-0.0596528231641327,0.0687058044588151],[0,0,0,0],[8.999999E+09,8.999999E+09,8.999999E+09,8.999999E+09,8.999999E+09,8.999999E+09]];
	LOCAL CONST Robtarget Tr_meulage_bavure_P402 :=[[169.97515625,-281.5585625,20],[0.750729470818659,-0.651001875374858,-0.0735449255704238,0.0848113425527227],[0,0,0,0],[8.999999E+09,8.999999E+09,8.999999E+09,8.999999E+09,8.999999E+09,8.999999E+09]];
	LOCAL CONST Robtarget Tr_meulage_bavure_P403 :=[[170.659125,-281.3914375,20],[0.748910458534829,-0.648620921391645,-0.0888630581532673,0.102603032732252],[0,0,0,0],[8.999999E+09,8.999999E+09,8.999999E+09,8.999999E+09,8.999999E+09,8.999999E+09]];
	LOCAL CONST Robtarget Tr_meulage_bavure_P404 :=[[171.2158125,-281.222375,20],[0.746418737945591,-0.645683191215672,-0.105394308580165,0.121837284704501],[0,0,0,0],[8.999999E+09,8.999999E+09,8.999999E+09,8.999999E+09,8.999999E+09,8.999999E+09]];
	LOCAL CONST Robtarget Tr_meulage_bavure_P405 :=[[173.825015625,-280.50290625,20],[0.7431896392694,-0.642155335382306,-0.122847849605117,0.142176267956559],[0,0,0,0],[8.999999E+09,8.999999E+09,8.999999E+09,8.999999E+09,8.999999E+09,8.999999E+09]];
	LOCAL CONST Robtarget Tr_meulage_bavure_P406 :=[[175.65253125,-279.8055,20],[0.739236883685868,-0.638016246665018,-0.140838688535754,0.163182605082216],[0,0,0,0],[8.999999E+09,8.999999E+09,8.999999E+09,8.999999E+09,8.999999E+09,8.999999E+09]];
	LOCAL CONST Robtarget Tr_meulage_bavure_P407 :=[[178.34278125,-278.7875625,20],[0.734593059919747,-0.633322649797811,-0.158975881050089,0.184396656193026],[0,0,0,0],[8.999999E+09,8.999999E+09,8.999999E+09,8.999999E+09,8.999999E+09,8.999999E+09]];
	LOCAL CONST Robtarget Tr_meulage_bavure_P408 :=[[179.2655625,-278.2315,20],[0.729343337910948,-0.628156620347567,-0.176895717735746,0.205390994946698],[0,0,0,0],[8.999999E+09,8.999999E+09,8.999999E+09,8.999999E+09,8.999999E+09,8.999999E+09]];
	LOCAL CONST Robtarget Tr_meulage_bavure_P409 :=[[180.78778125,-277.339875,20],[0.723615012545134,-0.622604651710126,-0.194295930689931,0.225818184842477],[0,0,0,0],[8.999999E+09,8.999999E+09,8.999999E+09,8.999999E+09,8.999999E+09,8.999999E+09]];
	LOCAL CONST Robtarget Tr_meulage_bavure_P410 :=[[181.82525,-276.6099375,20],[0.717525013517294,-0.616776400349876,-0.210969847350159,0.245431152174101],[0,0,0,0],[8.999999E+09,8.999999E+09,8.999999E+09,8.999999E+09,8.999999E+09,8.999999E+09]];
	LOCAL CONST Robtarget Tr_meulage_bavure_P411 :=[[182.823296875,-275.81684375,20],[0.711161676785787,-0.610765200116398,-0.226835501826781,0.264122310509727],[0,0,0,0],[8.999999E+09,8.999999E+09,8.999999E+09,8.999999E+09,8.999999E+09,8.999999E+09]];
	LOCAL CONST Robtarget Tr_meulage_bavure_P412 :=[[184.879875,-273.92253125,20],[0.704580934743856,-0.604636894677965,-0.241904484308205,0.281890319914044],[0,0,0,0],[8.999999E+09,8.999999E+09,8.999999E+09,8.999999E+09,8.999999E+09,8.999999E+09]];
	LOCAL CONST Robtarget Tr_meulage_bavure_P413 :=[[185.101140625,-273.6601875,20],[0.69781407118237,-0.598399020150575,-0.256262750192385,0.298836974965537],[0,0,0,0],[8.999999E+09,8.999999E+09,8.999999E+09,8.999999E+09,8.999999E+09,8.999999E+09]];
	LOCAL CONST Robtarget Tr_meulage_bavure_P414 :=[[185.19628125,-273.56965625,20],[0.690839787130852,-0.592038334984509,-0.270054183053407,0.315121780651744],[0,0,0,0],[8.999999E+09,8.999999E+09,8.999999E+09,8.999999E+09,8.999999E+09,8.999999E+09]];
	LOCAL CONST Robtarget Tr_meulage_bavure_P415 :=[[187.786375,-270.56334375,20],[0.683612188766417,-0.585514473250394,-0.283436797129505,0.330924098574387],[0,0,0,0],[8.999999E+09,8.999999E+09,8.999999E+09,8.999999E+09,8.999999E+09,8.999999E+09]];
	LOCAL CONST Robtarget Tr_meulage_bavure_P416 :=[[188.3231875,-270.1005625,20],[0.676065476231399,-0.578771164959462,-0.296566748409769,0.34642109375316],[0,0,0,0],[8.999999E+09,8.999999E+09,8.999999E+09,8.999999E+09,8.999999E+09,8.999999E+09]];
	LOCAL CONST Robtarget Tr_meulage_bavure_P417 :=[[189.5753125,-268.331875,20],[0.668134664286423,-0.571759701093499,-0.309563029526245,0.361742512479352],[0,0,0,0],[8.999999E+09,8.999999E+09,8.999999E+09,8.999999E+09,8.999999E+09,8.999999E+09]];
	LOCAL CONST Robtarget Tr_meulage_bavure_P418 :=[[190.4013125,-267.088625,20],[0.659760222688129,-0.564439530474089,-0.32251133994896,0.376975994727818],[0,0,0,0],[8.999999E+09,8.999999E+09,8.999999E+09,8.999999E+09,8.999999E+09,8.999999E+09]];
	LOCAL CONST Robtarget Tr_meulage_bavure_P419 :=[[191.06371875,-265.90546875,20],[0.650911737903026,-0.556786965804725,-0.335442287616095,0.392148767496357],[0,0,0,0],[8.999999E+09,8.999999E+09,8.999999E+09,8.999999E+09,8.999999E+09,8.999999E+09]];
	LOCAL CONST Robtarget Tr_meulage_bavure_P420 :=[[191.416015625,-264.96075,20],[0.641614615468793,-0.548800566891777,-0.34831198949455,0.407219082276907],[0,0,0,0],[8.999999E+09,8.999999E+09,8.999999E+09,8.999999E+09,8.999999E+09,8.999999E+09]];
	LOCAL CONST Robtarget Tr_meulage_bavure_P421 :=[[192.0755625,-262.849625,20],[0.63192816694281,-0.540535900227202,-0.361030213275699,0.422072170951807],[0,0,0,0],[8.999999E+09,8.999999E+09,8.999999E+09,8.999999E+09,8.999999E+09,8.999999E+09]];
	LOCAL CONST Robtarget Tr_meulage_bavure_P422 :=[[193.15484375,-259.811703125,20],[0.621946455479366,-0.532074466407673,-0.373482220150297,0.436566604248708],[0,0,0,0],[8.999999E+09,8.999999E+09,8.999999E+09,8.999999E+09,8.999999E+09,8.999999E+09]];
	LOCAL CONST Robtarget Tr_meulage_bavure_P423 :=[[193.31403125,-259.121703125,20],[0.611815915461986,-0.523536999852556,-0.38551480977315,0.450520395563141],[0,0,0,0],[8.999999E+09,8.999999E+09,8.999999E+09,8.999999E+09,8.999999E+09,8.999999E+09]];
	LOCAL CONST Robtarget Tr_meulage_bavure_P424 :=[[193.619015625,-258.479,20],[0.601707732722379,-0.515099933942939,-0.396971302455896,0.463717206345143],[0,0,0,0],[8.999999E+09,8.999999E+09,8.999999E+09,8.999999E+09,8.999999E+09,8.999999E+09]];
	LOCAL CONST Robtarget Tr_meulage_bavure_P425 :=[[194.224,-255.81478125,20],[0.591840301122901,-0.506910870768301,-0.407681398721124,0.475985613438542],[0,0,0,0],[8.999999E+09,8.999999E+09,8.999999E+09,8.999999E+09,8.999999E+09,8.999999E+09]];
	LOCAL CONST Robtarget Tr_meulage_bavure_P426 :=[[194.328,-254.526515625,20],[0.582430394636542,-0.499176098982662,-0.417497031776463,0.487128613474734],[0,0,0,0],[8.999999E+09,8.999999E+09,8.999999E+09,8.999999E+09,8.999999E+09,8.999999E+09]];
	LOCAL CONST Robtarget Tr_meulage_bavure_P427 :=[[194.56365625,-252.04003125,20],[0.573692827680917,-0.49206421616566,-0.426294926715048,0.497013060284899],[0,0,0,0],[8.999999E+09,8.999999E+09,8.999999E+09,8.999999E+09,8.999999E+09,8.999999E+09]];
	LOCAL CONST Robtarget Tr_meulage_bavure_P428 :=[[194.570375,-250.342390625,20],[0.565786527162031,-0.485728856484631,-0.434016984511458,0.505551521425503],[0,0,0,0],[8.999999E+09,8.999999E+09,8.999999E+09,8.999999E+09,8.999999E+09,8.999999E+09]];
	LOCAL CONST Robtarget Tr_meulage_bavure_P429 :=[[194.728703125,-248.301890625,20],[0.558855149659692,-0.480257358705545,-0.440617540934349,0.512727972446387],[0,0,0,0],[8.999999E+09,8.999999E+09,8.999999E+09,8.999999E+09,8.999999E+09,8.999999E+09]];
	LOCAL CONST Robtarget Tr_meulage_bavure_P430 :=[[194.732234375,-248.171671875,20],[0.55294525989914,-0.475723884432231,-0.44613703440684,0.518555755793388],[0,0,0,0],[8.999999E+09,8.999999E+09,8.999999E+09,8.999999E+09,8.999999E+09,8.999999E+09]];
	LOCAL CONST Robtarget Tr_meulage_bavure_P431 :=[[194.597171875,-246.789203125,20],[0.548073220478166,-0.472118469491783,-0.450625244778318,0.523122150676024],[0,0,0,0],[8.999999E+09,8.999999E+09,8.999999E+09,8.999999E+09,8.999999E+09,8.999999E+09]];
	LOCAL CONST Robtarget Tr_meulage_bavure_P432 :=[[194.593140625,-243.63484375,20],[0.544183240774223,-0.469410257574642,-0.454184003729118,0.526531576736629],[0,0,0,0],[8.999999E+09,8.999999E+09,8.999999E+09,8.999999E+09,8.999999E+09,8.999999E+09]];
	LOCAL CONST Robtarget Tr_meulage_bavure_P433 :=[[194.543328125,-239.444046875,20],[0.541175990991956,-0.467512859540277,-0.456936032193781,0.528932637886292],[0,0,0,0],[8.999999E+09,8.999999E+09,8.999999E+09,8.999999E+09,8.999999E+09,8.999999E+09]];
	LOCAL CONST Robtarget Tr_meulage_bavure_P434 :=[[194.5338125,-237.029953125,20],[0.538923123934595,-0.466327716639694,-0.459017337239009,0.530474703728836],[0,0,0,0],[8.999999E+09,8.999999E+09,8.999999E+09,8.999999E+09,8.999999E+09,8.999999E+09]];
	LOCAL CONST Robtarget Tr_meulage_bavure_P435 :=[[194.621640625,-229.919,20],[0.537306281316416,-0.465726946156977,-0.46054003270627,0.531322171526964],[0,0,0,0],[8.999999E+09,8.999999E+09,8.999999E+09,8.999999E+09,8.999999E+09,8.999999E+09]];
	LOCAL CONST Robtarget Tr_meulage_bavure_P436 :=[[194.56628125,-227.704625,20],[0.536176871230432,-0.465589985761751,-0.461640217480401,0.531628288864095],[0,0,0,0],[8.999999E+09,8.999999E+09,8.999999E+09,8.999999E+09,8.999999E+09,8.999999E+09]];
	LOCAL CONST Robtarget Tr_meulage_bavure_P437 :=[[194.584171875,-225.601953125,20],[0.53541807854372,-0.46582468491876,-0.462422468672965,0.531507577138172],[0,0,0,0],[8.999999E+09,8.999999E+09,8.999999E+09,8.999999E+09,8.999999E+09,8.999999E+09]];
	LOCAL CONST Robtarget Tr_meulage_bavure_P438 :=[[194.47778125,-220.538453125,20],[0.534939080384706,-0.466335066342682,-0.462963328673649,0.531071315813372],[0,0,0,0],[8.999999E+09,8.999999E+09,8.999999E+09,8.999999E+09,8.999999E+09,8.999999E+09]];
	LOCAL CONST Robtarget Tr_meulage_bavure_P439 :=[[194.495359375,-217.15465625,20],[0.534662278677667,-0.467065631461937,-0.463330907165906,0.530387041820485],[0,0,0,0],[8.999999E+09,8.999999E+09,8.999999E+09,8.999999E+09,8.999999E+09,8.999999E+09]];
	LOCAL CONST Robtarget Tr_meulage_bavure_P440 :=[[194.646796875,-215.308078125,20],[0.534555829030241,-0.467973369395183,-0.463549459495934,0.529502492711544],[0,0,0,0],[8.999999E+09,8.999999E+09,8.999999E+09,8.999999E+09,8.999999E+09,8.999999E+09]];
	LOCAL CONST Robtarget Tr_meulage_bavure_P441 :=[[194.65746875,-214.213546875,20],[0.534569025704571,-0.469037914153703,-0.463664800974882,0.528445213982047],[0,0,0,0],[8.999999E+09,8.999999E+09,8.999999E+09,8.999999E+09,8.999999E+09,8.999999E+09]];
	LOCAL CONST Robtarget Tr_meulage_bavure_P442 :=[[194.5858125,-210.38871875,20],[0.534713290763085,-0.470240602703531,-0.463661377773904,0.527232016299406],[0,0,0,0],[8.999999E+09,8.999999E+09,8.999999E+09,8.999999E+09,8.999999E+09,8.999999E+09]];
	LOCAL CONST Robtarget Tr_meulage_bavure_P443 :=[[194.489375,-208.452984375,20],[0.534988625629728,-0.471576074683865,-0.463536482613058,0.525867954451768],[0,0,0,0],[8.999999E+09,8.999999E+09,8.999999E+09,8.999999E+09,8.999999E+09,8.999999E+09]];
	LOCAL CONST Robtarget Tr_meulage_bavure_P444 :=[[194.51184375,-202.228609375,20],[0.535375881948296,-0.473045920691513,-0.463307004656784,0.524353736881088],[0,0,0,0],[8.999999E+09,8.999999E+09,8.999999E+09,8.999999E+09,8.999999E+09,8.999999E+09]];
	LOCAL CONST Robtarget Tr_meulage_bavure_P445 :=[[194.543890625,-198.23209375,20],[0.535881469168044,-0.474613622237328,-0.462960551156864,0.522724103769468],[0,0,0,0],[8.999999E+09,8.999999E+09,8.999999E+09,8.999999E+09,8.999999E+09,8.999999E+09]];
	LOCAL CONST Robtarget Tr_meulage_bavure_P446 :=[[194.68871875,-191.811140625,20],[0.53642931962327,-0.476252218305106,-0.462568265397518,0.521016323597555],[0,0,0,0],[8.999999E+09,8.999999E+09,8.999999E+09,8.999999E+09,8.999999E+09,8.999999E+09]];
	LOCAL CONST Robtarget Tr_meulage_bavure_P447 :=[[194.711125,-190.693,20],[0.536950883653265,-0.477891966154174,-0.462191037960668,0.519309600968552],[0,0,0,0],[8.999999E+09,8.999999E+09,8.999999E+09,8.999999E+09,8.999999E+09,8.999999E+09]];
	LOCAL CONST Robtarget Tr_meulage_bavure_P448 :=[[194.798640625,-190.142390625,20],[0.53736383596968,-0.479429914333024,-0.461902874163417,0.517718842494799],[0,0,0,0],[8.999999E+09,8.999999E+09,8.999999E+09,8.999999E+09,8.999999E+09,8.999999E+09]];
	LOCAL CONST Robtarget Tr_meulage_bavure_P449 :=[[194.829953125,-188.23275,20],[0.537524685186614,-0.480739474344179,-0.46183955099412,0.516392292506253],[0,0,0,0],[8.999999E+09,8.999999E+09,8.999999E+09,8.999999E+09,8.999999E+09,8.999999E+09]];
	LOCAL CONST Robtarget Tr_meulage_bavure_P450 :=[[194.733453125,-187.422015625,20],[0.537277924770666,-0.481680649196569,-0.462150264920267,0.515493274813382],[0,0,0,0],[8.999999E+09,8.999999E+09,8.999999E+09,8.999999E+09,8.999999E+09,8.999999E+09]];
	LOCAL CONST Robtarget Tr_meulage_bavure_P451 :=[[194.835203125,-182.75234375,20],[0.536484529085605,-0.482101639339727,-0.462967823508539,0.515192346404244],[0,0,0,0],[8.999999E+09,8.999999E+09,8.999999E+09,8.999999E+09,8.999999E+09,8.999999E+09]];
	LOCAL CONST Robtarget Tr_meulage_bavure_P452 :=[[194.830015625,-180.5726875,20],[0.534988014854943,-0.481880124416652,-0.464442348957787,0.515628426435484],[0,0,0,0],[8.999999E+09,8.999999E+09,8.999999E+09,8.999999E+09,8.999999E+09,8.999999E+09]];
	LOCAL CONST Robtarget Tr_meulage_bavure_P453 :=[[195.242125,-177.5310625,20],[0.532697322537403,-0.480910040095103,-0.466654585703072,0.516906755169153],[0,0,0,0],[8.999999E+09,8.999999E+09,8.999999E+09,8.999999E+09,8.999999E+09,8.999999E+09]];
	LOCAL CONST Robtarget Tr_meulage_bavure_P454 :=[[195.2629375,-176.968890625,20],[0.529549116065891,-0.479142660793729,-0.469653789332793,0.519062002507107],[0,0,0,0],[8.999999E+09,8.999999E+09,8.999999E+09,8.999999E+09,8.999999E+09,8.999999E+09]];
	LOCAL CONST Robtarget Tr_meulage_bavure_P455 :=[[195.54271875,-174.069734375,20],[0.525582989428987,-0.476583693008104,-0.473382749280895,0.522052945078283],[0,0,0,0],[8.999999E+09,8.999999E+09,8.999999E+09,8.999999E+09,8.999999E+09,8.999999E+09]];
	LOCAL CONST Robtarget Tr_meulage_bavure_P456 :=[[195.546078125,-173.54875,20],[0.52093390410091,-0.473342074133671,-0.477693293166649,0.525722613244495],[0,0,0,0],[8.999999E+09,8.999999E+09,8.999999E+09,8.999999E+09,8.999999E+09,8.999999E+09]];
	LOCAL CONST Robtarget Tr_meulage_bavure_P457 :=[[195.765015625,-170.15915625,20],[0.515799344362131,-0.469619195240062,-0.482386794671815,0.529822449641315],[0,0,0,0],[8.999999E+09,8.999999E+09,8.999999E+09,8.999999E+09,8.999999E+09,8.999999E+09]];
	LOCAL CONST Robtarget Tr_meulage_bavure_P458 :=[[195.752625,-170.050484375,20],[0.510525014924896,-0.465700443861927,-0.48713806065568,0.534026043918611],[0,0,0,0],[8.999999E+09,8.999999E+09,8.999999E+09,8.999999E+09,8.999999E+09,8.999999E+09]];
	LOCAL CONST Robtarget Tr_meulage_bavure_P459 :=[[195.773625,-169.830234375,20],[0.505510972167725,-0.461947298861148,-0.491596190929011,0.537955885883795],[0,0,0,0],[8.999999E+09,8.999999E+09,8.999999E+09,8.999999E+09,8.999999E+09,8.999999E+09]];
	LOCAL CONST Robtarget Tr_meulage_bavure_P460 :=[[195.72803125,-166.663625,20],[0.501176010418104,-0.458764722828578,-0.495418862577135,0.541218704658466],[0,0,0,0],[8.999999E+09,8.999999E+09,8.999999E+09,8.999999E+09,8.999999E+09,8.999999E+09]];
	LOCAL CONST Robtarget Tr_meulage_bavure_P461 :=[[195.647703125,-165.5805625,20],[0.497952859603593,-0.456523327977337,-0.498259529466621,0.54347662499946],[0,0,0,0],[8.999999E+09,8.999999E+09,8.999999E+09,8.999999E+09,8.999999E+09,8.999999E+09]];
	LOCAL CONST Robtarget Tr_meulage_bavure_P462 :=[[195.45025,-163.247515625,20],[0.496131491160969,-0.455515459845291,-0.499903532611418,0.544477425981052],[0,0,0,0],[8.999999E+09,8.999999E+09,8.999999E+09,8.999999E+09,8.999999E+09,8.999999E+09]];
	LOCAL CONST Robtarget Tr_meulage_bavure_P463 :=[[195.419859375,-163.121234375,20],[0.495856230007745,-0.455862428194855,-0.500240751184346,0.544127959745975],[0,0,0,0],[8.999999E+09,8.999999E+09,8.999999E+09,8.999999E+09,8.999999E+09,8.999999E+09]];
	LOCAL CONST Robtarget Tr_meulage_bavure_P464 :=[[195.417546875,-163.012921875,20],[0.497082647301519,-0.457531941805984,-0.499303962013586,0.542465591071448],[0,0,0,0],[8.999999E+09,8.999999E+09,8.999999E+09,8.999999E+09,8.999999E+09,8.999999E+09]];
	LOCAL CONST Robtarget Tr_meulage_bavure_P465 :=[[195.095640625,-159.529234375,20],[0.49957529068319,-0.460308783539173,-0.497269156315943,0.539688557329432],[0,0,0,0],[8.999999E+09,8.999999E+09,8.999999E+09,8.999999E+09,8.999999E+09,8.999999E+09]];
	LOCAL CONST Robtarget Tr_meulage_bavure_P466 :=[[195.095765625,-159.4821875,20],[0.502947570344507,-0.463849979891408,-0.494437981204636,0.536113812899447],[0,0,0,0],[8.999999E+09,8.999999E+09,8.999999E+09,8.999999E+09,8.999999E+09,8.999999E+09]];
	LOCAL CONST Robtarget Tr_meulage_bavure_P467 :=[[195.417484375,-155.614375,20],[0.506774591329933,-0.467735043146827,-0.49114906893713,0.532142870925662],[0,0,0,0],[8.999999E+09,8.999999E+09,8.999999E+09,8.999999E+09,8.999999E+09,8.999999E+09]];
	LOCAL CONST Robtarget Tr_meulage_bavure_P468 :=[[195.9191875,-152.753203125,20],[0.510594535971404,-0.471557575725654,-0.487800979169961,0.528182617408712],[0,0,0,0],[8.999999E+09,8.999999E+09,8.999999E+09,8.999999E+09,8.999999E+09,8.999999E+09]];
	LOCAL CONST Robtarget Tr_meulage_bavure_P469 :=[[195.984125,-151.866359375,20],[0.514058793193058,-0.47497803151457,-0.4847097156986,0.524591191526148],[0,0,0,0],[8.999999E+09,8.999999E+09,8.999999E+09,8.999999E+09,8.999999E+09,8.999999E+09]];
	LOCAL CONST Robtarget Tr_meulage_bavure_P470 :=[[195.95934375,-149.530234375,20],[0.516915992487683,-0.477785014020894,-0.482123251654328,0.521609535286487],[0,0,0,0],[8.999999E+09,8.999999E+09,8.999999E+09,8.999999E+09,8.999999E+09,8.999999E+09]];
	LOCAL CONST Robtarget Tr_meulage_bavure_P471 :=[[195.903375,-147.17734375,20],[0.519058152047249,-0.479863009685189,-0.480160738738845,0.519380199567651],[0,0,0,0],[8.999999E+09,8.999999E+09,8.999999E+09,8.999999E+09,8.999999E+09,8.999999E+09]];
	LOCAL CONST Robtarget Tr_meulage_bavure_P472 :=[[195.892390625,-144.2560625,20],[0.520501525869182,-0.48122774792076,-0.478825694722378,0.517903437208712],[0,0,0,0],[8.999999E+09,8.999999E+09,8.999999E+09,8.999999E+09,8.999999E+09,8.999999E+09]];
	LOCAL CONST Robtarget Tr_meulage_bavure_P473 :=[[195.81928125,-141.7416875,20],[0.521320316606221,-0.481949739234577,-0.478061224323266,0.51711414807937],[0,0,0,0],[8.999999E+09,8.999999E+09,8.999999E+09,8.999999E+09,8.999999E+09,8.999999E+09]];
	LOCAL CONST Robtarget Tr_meulage_bavure_P474 :=[[195.647578125,-136.490859375,20],[0.521655050459169,-0.482149037371728,-0.477741428914296,0.516886294257146],[0,0,0,0],[8.999999E+09,8.999999E+09,8.999999E+09,8.999999E+09,8.999999E+09,8.999999E+09]];
	LOCAL CONST Robtarget Tr_meulage_bavure_P475 :=[[195.674625,-135.26503125,20],[0.521668559930331,-0.481971309158619,-0.477715561918344,0.517062290859798],[0,0,0,0],[8.999999E+09,8.999999E+09,8.999999E+09,8.999999E+09,8.999999E+09,8.999999E+09]];
	LOCAL CONST Robtarget Tr_meulage_bavure_P476 :=[[195.55103125,-133.268390625,20],[0.521476844567545,-0.48156260728371,-0.477877684181738,0.517486497221996],[0,0,0,0],[8.999999E+09,8.999999E+09,8.999999E+09,8.999999E+09,8.999999E+09,8.999999E+09]];
	LOCAL CONST Robtarget Tr_meulage_bavure_P477 :=[[195.547125,-130.4526796875,20],[0.521206529655309,-0.481022137920399,-0.478107752901303,0.51804867810933],[0,0,0,0],[8.999999E+09,8.999999E+09,8.999999E+09,8.999999E+09,8.999999E+09,8.999999E+09]];
	LOCAL CONST Robtarget Tr_meulage_bavure_P478 :=[[195.559453125,-126.6521015625,20],[0.520948133773278,-0.480435682697267,-0.478321226769846,0.518655377616717],[0,0,0,0],[8.999999E+09,8.999999E+09,8.999999E+09,8.999999E+09,8.999999E+09,8.999999E+09]];
	LOCAL CONST Robtarget Tr_meulage_bavure_P479 :=[[195.469421875,-124.897171875,20],[0.520748375679681,-0.479852131184057,-0.478475071016483,0.519253953129743],[0,0,0,0],[8.999999E+09,8.999999E+09,8.999999E+09,8.999999E+09,8.999999E+09,8.999999E+09]];
	LOCAL CONST Robtarget Tr_meulage_bavure_P480 :=[[195.467953125,-122.5718203125,20],[0.520642414482296,-0.479298370071215,-0.478536458619034,0.519814780918622],[0,0,0,0],[8.999999E+09,8.999999E+09,8.999999E+09,8.999999E+09,8.999999E+09,8.999999E+09]];
	LOCAL CONST Robtarget Tr_meulage_bavure_P481 :=[[195.35809375,-117.9137421875,20],[0.520641635606473,-0.478774291139471,-0.478494256959886,0.520337113296101],[0,0,0,0],[8.999999E+09,8.999999E+09,8.999999E+09,8.999999E+09,8.999999E+09,8.999999E+09]];
	LOCAL CONST Robtarget Tr_meulage_bavure_P482 :=[[195.3308125,-113.6826796875,20],[0.520724250959249,-0.478278830334483,-0.478370300262356,0.520823838494084],[0,0,0,0],[8.999999E+09,8.999999E+09,8.999999E+09,8.999999E+09,8.999999E+09,8.999999E+09]];
	LOCAL CONST Robtarget Tr_meulage_bavure_P483 :=[[195.35315625,-108.728484375,20],[0.520877360960489,-0.477813665640887,-0.4781777796674,0.521274291326564],[0,0,0,0],[8.999999E+09,8.999999E+09,8.999999E+09,8.999999E+09,8.999999E+09,8.999999E+09]];
	LOCAL CONST Robtarget Tr_meulage_bavure_P484 :=[[195.430546875,-104.731625,20],[0.521074319103518,-0.477365489043257,-0.477942250417734,0.52170389025474],[0,0,0,0],[8.999999E+09,8.999999E+09,8.999999E+09,8.999999E+09,8.999999E+09,8.999999E+09]];
	LOCAL CONST Robtarget Tr_meulage_bavure_P485 :=[[195.3384375,-100.7190859375,20],[0.521313096895726,-0.47691233951396,-0.477663854357816,0.522134578115971],[0,0,0,0],[8.999999E+09,8.999999E+09,8.999999E+09,8.999999E+09,8.999999E+09,8.999999E+09]];
	LOCAL CONST Robtarget Tr_meulage_bavure_P486 :=[[195.439390625,-94.93809375,20],[0.521564934475831,-0.476446019550349,-0.477370468496382,0.52257692772203],[0,0,0,0],[8.999999E+09,8.999999E+09,8.999999E+09,8.999999E+09,8.999999E+09,8.999999E+09]];
	LOCAL CONST Robtarget Tr_meulage_bavure_P487 :=[[195.470890625,-91.3452421875,20],[0.521818184713322,-0.475949608069517,-0.477072033419719,0.523048781290751],[0,0,0,0],[8.999999E+09,8.999999E+09,8.999999E+09,8.999999E+09,8.999999E+09,8.999999E+09]];
	LOCAL CONST Robtarget Tr_meulage_bavure_P488 :=[[195.4794375,-89.6339140625,20],[0.52208501164977,-0.47541460070228,-0.476755447365934,0.523557486296069],[0,0,0,0],[8.999999E+09,8.999999E+09,8.999999E+09,8.999999E+09,8.999999E+09,8.999999E+09]];
	LOCAL CONST Robtarget Tr_meulage_bavure_P489 :=[[195.3746875,-88.54171875,20],[0.522336951157636,-0.474869123837209,-0.476451578552151,0.524077587744974],[0,0,0,0],[8.999999E+09,8.999999E+09,8.999999E+09,8.999999E+09,8.999999E+09,8.999999E+09]];
	LOCAL CONST Robtarget Tr_meulage_bavure_P490 :=[[195.357421875,-87.078109375,20],[0.522592800634613,-0.474307412556428,-0.476141065567559,0.524613122976434],[0,0,0,0],[8.999999E+09,8.999999E+09,8.999999E+09,8.999999E+09,8.999999E+09,8.999999E+09]];
	LOCAL CONST Robtarget Tr_meulage_bavure_P491 :=[[195.35925,-79.8096796875,20],[0.522859252066815,-0.473748912181814,-0.47581914250538,0.525144089141375],[0,0,0,0],[8.999999E+09,8.999999E+09,8.999999E+09,8.999999E+09,8.999999E+09,8.999999E+09]];
	LOCAL CONST Robtarget Tr_meulage_bavure_P492 :=[[195.392578125,-78.691890625,20],[0.523160670734168,-0.473208851713561,-0.475463189314836,0.525652975701148],[0,0,0,0],[8.999999E+09,8.999999E+09,8.999999E+09,8.999999E+09,8.999999E+09,8.999999E+09]];
	LOCAL CONST Robtarget Tr_meulage_bavure_P493 :=[[195.510859375,-76.4956640625,20],[0.523514936901914,-0.472724747165125,-0.475059556178352,0.526100600970842],[0,0,0,0],[8.999999E+09,8.999999E+09,8.999999E+09,8.999999E+09,8.999999E+09,8.999999E+09]];
	LOCAL CONST Robtarget Tr_meulage_bavure_P494 :=[[195.567875,-73.871859375,20],[0.523966496969294,-0.472315885107119,-0.474566461730044,0.526463187820603],[0,0,0,0],[8.999999E+09,8.999999E+09,8.999999E+09,8.999999E+09,8.999999E+09,8.999999E+09]];
	LOCAL CONST Robtarget Tr_meulage_bavure_P495 :=[[195.536984375,-70.1845703125,20],[0.52455302043267,-0.47202777818378,-0.473951819133447,0.526691160470672],[0,0,0,0],[8.999999E+09,8.999999E+09,8.999999E+09,8.999999E+09,8.999999E+09,8.999999E+09]];
	LOCAL CONST Robtarget Tr_meulage_bavure_P496 :=[[195.6665,-64.1988515625,20],[0.525323870438147,-0.471918755117929,-0.473173385779295,0.526720482519891],[0,0,0,0],[8.999999E+09,8.999999E+09,8.999999E+09,8.999999E+09,8.999999E+09,8.999999E+09]];
	LOCAL CONST Robtarget Tr_meulage_bavure_P497 :=[[195.588875,-60.24858203125,20],[0.526329303245848,-0.472029378107555,-0.472185863610263,0.526503790066856],[0,0,0,0],[8.999999E+09,8.999999E+09,8.999999E+09,8.999999E+09,8.999999E+09,8.999999E+09]];
	LOCAL CONST Robtarget Tr_meulage_bavure_P498 :=[[195.70959375,-59.0367109375,20],[0.527613299881597,-0.472398895034946,-0.470949427253796,0.525994417011374],[0,0,0,0],[8.999999E+09,8.999999E+09,8.999999E+09,8.999999E+09,8.999999E+09,8.999999E+09]];
	LOCAL CONST Robtarget Tr_meulage_bavure_P499 :=[[195.76403125,-54.11868359375,20],[0.529229918278125,-0.473082411866549,-0.469414840506941,0.525127063379617],[0,0,0,0],[8.999999E+09,8.999999E+09,8.999999E+09,8.999999E+09,8.999999E+09,8.999999E+09]];
	LOCAL CONST Robtarget Tr_meulage_bavure_P500 :=[[195.733828125,-47.72703515625,20],[0.531180312145718,-0.474094857861161,-0.46757961048819,0.52388056806308],[0,0,0,0],[8.999999E+09,8.999999E+09,8.999999E+09,8.999999E+09,8.999999E+09,8.999999E+09]];
	LOCAL CONST Robtarget Tr_meulage_bavure_P501 :=[[195.62640625,-43.5126328125,20],[0.533466812714583,-0.47541744586906,-0.465435204089281,0.522265720385565],[0,0,0,0],[8.999999E+09,8.999999E+09,8.999999E+09,8.999999E+09,8.999999E+09,8.999999E+09]];
	LOCAL CONST Robtarget Tr_meulage_bavure_P502 :=[[195.73821875,-37.6500859375,20],[0.536068100955058,-0.47706331347887,-0.462998334428803,0.520263518216638],[0,0,0,0],[8.999999E+09,8.999999E+09,8.999999E+09,8.999999E+09,8.999999E+09,8.999999E+09]];
	LOCAL CONST Robtarget Tr_meulage_bavure_P503 :=[[195.921453125,-32.086853515625,20],[0.538930283730616,-0.47893983115253,-0.460307958174762,0.517964642668402],[0,0,0,0],[8.999999E+09,8.999999E+09,8.999999E+09,8.999999E+09,8.999999E+09,8.999999E+09]];
	LOCAL CONST Robtarget Tr_meulage_bavure_P504 :=[[195.960625,-29.015564453125,20],[0.541941641518877,-0.48098102635933,-0.457464320809651,0.515444375909094],[0,0,0,0],[8.999999E+09,8.999999E+09,8.999999E+09,8.999999E+09,8.999999E+09,8.999999E+09]];
	LOCAL CONST Robtarget Tr_meulage_bavure_P505 :=[[196.08875,-27.47216796875,20],[0.544958306115189,-0.483063506900514,-0.454598107689841,0.512845642841837],[0,0,0,0],[8.999999E+09,8.999999E+09,8.999999E+09,8.999999E+09,8.999999E+09,8.999999E+09]];
	LOCAL CONST Robtarget Tr_meulage_bavure_P506 :=[[196.117,-24.58123828125,20],[0.547843323014303,-0.485061020109299,-0.451837624011944,0.510319764193406],[0,0,0,0],[8.999999E+09,8.999999E+09,8.999999E+09,8.999999E+09,8.999999E+09,8.999999E+09]];
	LOCAL CONST Robtarget Tr_meulage_bavure_P507 :=[[196.22503125,-21.208283203125,20],[0.550452226407156,-0.486860993578157,-0.449324057314654,0.508012412145404],[0,0,0,0],[8.999999E+09,8.999999E+09,8.999999E+09,8.999999E+09,8.999999E+09,8.999999E+09]];
	LOCAL CONST Robtarget Tr_meulage_bavure_P508 :=[[196.336734375,-18.125548828125,20],[0.552667787930494,-0.488343455341004,-0.447174967333296,0.506076609220471],[0,0,0,0],[8.999999E+09,8.999999E+09,8.999999E+09,8.999999E+09,8.999999E+09,8.999999E+09]];
	LOCAL CONST Robtarget Tr_meulage_bavure_P509 :=[[196.5780625,-14.79180859375,20],[0.554436714827431,-0.489486580801952,-0.445449726053797,0.504556595462568],[0,0,0,0],[8.999999E+09,8.999999E+09,8.999999E+09,8.999999E+09,8.999999E+09,8.999999E+09]];
	LOCAL CONST Robtarget Tr_meulage_bavure_P510 :=[[196.6535625,-13.56756640625,20],[0.55574334696351,-0.490261196886437,-0.444169083728715,0.503494901853899],[0,0,0,0],[8.999999E+09,8.999999E+09,8.999999E+09,8.999999E+09,8.999999E+09,8.999999E+09]];
	LOCAL CONST Robtarget Tr_meulage_bavure_P511 :=[[197.05103125,-11.778259765625,20],[0.556663064724401,-0.490733347720341,-0.44326393535475,0.502816166626179],[0,0,0,0],[8.999999E+09,8.999999E+09,8.999999E+09,8.999999E+09,8.999999E+09,8.999999E+09]];
	LOCAL CONST Robtarget Tr_meulage_bavure_P512 :=[[197.165765625,-10.6510009765625,20],[0.557318805154766,-0.491043874307301,-0.442617209373985,0.502356117601972],[0,0,0,0],[8.999999E+09,8.999999E+09,8.999999E+09,8.999999E+09,8.999999E+09,8.999999E+09]];
	LOCAL CONST Robtarget Tr_meulage_bavure_P513 :=[[197.46465625,-8.638,20],[0.55786222230628,-0.491311252703207,-0.442081040985391,0.50196349179196],[0,0,0,0],[8.999999E+09,8.999999E+09,8.999999E+09,8.999999E+09,8.999999E+09,8.999999E+09]];
	LOCAL CONST Robtarget Tr_meulage_bavure_P514 :=[[197.80071875,-5.5700986328125,20],[0.558461943523774,-0.491674745891044,-0.441490174893773,0.501460494317242],[0,0,0,0],[8.999999E+09,8.999999E+09,8.999999E+09,8.999999E+09,8.999999E+09,8.999999E+09]];
	LOCAL CONST Robtarget Tr_meulage_bavure_P515 :=[[197.786859375,-4.8630068359375,20],[0.559278826100568,-0.492293204205487,-0.440686256972879,0.500649796448475],[0,0,0,0],[8.999999E+09,8.999999E+09,8.999999E+09,8.999999E+09,8.999999E+09,8.999999E+09]];
	LOCAL CONST Robtarget Tr_meulage_bavure_P516 :=[[197.737484375,-4.084716796875,20],[0.560414680217775,-0.493251676158857,-0.439566299803076,0.499419301029024],[0,0,0,0],[8.999999E+09,8.999999E+09,8.999999E+09,8.999999E+09,8.999999E+09,8.999999E+09]];
	LOCAL CONST Robtarget Tr_meulage_bavure_P517 :=[[197.739875,-3.37152099609375,20],[0.561893283206414,-0.494546284964603,-0.438101546573543,0.497761936275863],[0,0,0,0],[8.999999E+09,8.999999E+09,8.999999E+09,8.999999E+09,8.999999E+09,8.999999E+09]];
	LOCAL CONST Robtarget Tr_meulage_bavure_P518 :=[[197.066046875,5.1211240234375,20],[0.563633683262902,-0.496132912434835,-0.436366237778737,0.495735525070833],[0,0,0,0],[8.999999E+09,8.999999E+09,8.999999E+09,8.999999E+09,8.999999E+09,8.999999E+09]];
	LOCAL CONST Robtarget Tr_meulage_bavure_P519 :=[[197.23859375,8.1240234375,20],[0.565465602404964,-0.497861749102969,-0.434525008884909,0.493528467193629],[0,0,0,0],[8.999999E+09,8.999999E+09,8.999999E+09,8.999999E+09,8.999999E+09,8.999999E+09]];
	LOCAL CONST Robtarget Tr_meulage_bavure_P520 :=[[197.0181875,19.5517265625,20],[0.567204819638098,-0.499574062282659,-0.432761339168221,0.491347201269167],[0,0,0,0],[8.999999E+09,8.999999E+09,8.999999E+09,8.999999E+09,8.999999E+09,8.999999E+09]];
	LOCAL CONST Robtarget Tr_meulage_bavure_P521 :=[[197.008609375,21.261322265625,20],[0.56862367193101,-0.501055907659082,-0.431309227725694,0.489471599991556],[0,0,0,0],[8.999999E+09,8.999999E+09,8.999999E+09,8.999999E+09,8.999999E+09,8.999999E+09]];
	LOCAL CONST Robtarget Tr_meulage_bavure_P522 :=[[197.145453125,25.0752265625,20],[0.569510363173597,-0.502129354482035,-0.43039187036304,0.488146387399042],[0,0,0,0],[8.999999E+09,8.999999E+09,8.999999E+09,8.999999E+09,8.999999E+09,8.999999E+09]];
	LOCAL CONST Robtarget Tr_meulage_bavure_P523 :=[[197.38690625,29.263123046875,20],[0.569723086389396,-0.502672556001333,-0.430162424567986,0.487540967271284],[0,0,0,0],[8.999999E+09,8.999999E+09,8.999999E+09,8.999999E+09,8.999999E+09,8.999999E+09]];
	LOCAL CONST Robtarget Tr_meulage_bavure_P524 :=[[197.388,31.528595703125,20],[0.569179355974741,-0.502586395277889,-0.430711030268148,0.4877804674432],[0,0,0,0],[8.999999E+09,8.999999E+09,8.999999E+09,8.999999E+09,8.999999E+09,8.999999E+09]];
	LOCAL CONST Robtarget Tr_meulage_bavure_P525 :=[[198.2240625,34.22537109375,20],[0.567882487652613,-0.501893528537537,-0.432032257317222,0.488835856773013],[0,0,0,0],[8.999999E+09,8.999999E+09,8.999999E+09,8.999999E+09,8.999999E+09,8.999999E+09]];
	LOCAL CONST Robtarget Tr_meulage_bavure_P526 :=[[198.098875,36.28469921875,20],[0.565955950312789,-0.500692973849385,-0.433992726397454,0.490561639019514],[0,0,0,0],[8.999999E+09,8.999999E+09,8.999999E+09,8.999999E+09,8.999999E+09,8.999999E+09]];
	LOCAL CONST Robtarget Tr_meulage_bavure_P527 :=[[198.0910625,36.85760546875,20],[0.563576109088941,-0.499143298932488,-0.436403372200435,0.492737286114062],[0,0,0,0],[8.999999E+09,8.999999E+09,8.999999E+09,8.999999E+09,8.999999E+09,8.999999E+09]];
	LOCAL CONST Robtarget Tr_meulage_bavure_P528 :=[[198.2185625,37.84982421875,20],[0.561007714082136,-0.497455190933396,-0.438989447696362,0.495072663924195],[0,0,0,0],[8.999999E+09,8.999999E+09,8.999999E+09,8.999999E+09,8.999999E+09,8.999999E+09]];
	LOCAL CONST Robtarget Tr_meulage_bavure_P529 :=[[198.25421875,39.7279375,20],[0.55854978005346,-0.495935862225051,-0.441449440739616,0.49718422645133],[0,0,0,0],[8.999999E+09,8.999999E+09,8.999999E+09,8.999999E+09,8.999999E+09,8.999999E+09]];
	LOCAL CONST Robtarget Tr_meulage_bavure_P530 :=[[198.3125,47.5269453125,20],[0.556498599204347,-0.494799469960441,-0.443493418918168,0.498794928790119],[0,0,0,0],[8.999999E+09,8.999999E+09,8.999999E+09,8.999999E+09,8.999999E+09,8.999999E+09]];
	LOCAL CONST Robtarget Tr_meulage_bavure_P531 :=[[198.5131875,54.620453125,20],[0.555096252594281,-0.494277805789633,-0.444889419659799,0.499630869076701],[0,0,0,0],[8.999999E+09,8.999999E+09,8.999999E+09,8.999999E+09,8.999999E+09,8.999999E+09]];
	LOCAL CONST Robtarget Tr_meulage_bavure_P532 :=[[198.424375,57.57684375,20],[0.554447735674805,-0.494460831334473,-0.445539105266947,0.499590933023242],[0,0,0,0],[8.999999E+09,8.999999E+09,8.999999E+09,8.999999E+09,8.999999E+09,8.999999E+09]];
	LOCAL CONST Robtarget Tr_meulage_bavure_P533 :=[[198.384703125,57.87515234375,20],[0.554507376392116,-0.495321081759878,-0.445486852647339,0.498718417154735],[0,0,0,0],[8.999999E+09,8.999999E+09,8.999999E+09,8.999999E+09,8.999999E+09,8.999999E+09]];
	LOCAL CONST Robtarget Tr_meulage_bavure_P534 :=[[196.961484375,65.591671875,20],[0.555126255473963,-0.496709575809969,-0.444873627182897,0.497194020096048],[0,0,0,0],[8.999999E+09,8.999999E+09,8.999999E+09,8.999999E+09,8.999999E+09,8.999999E+09]];
	LOCAL CONST Robtarget Tr_meulage_bavure_P535 :=[[196.946046875,67.0342109375,20],[0.555988490928653,-0.498353690922051,-0.444007017795409,0.49535660371865],[0,0,0,0],[8.999999E+09,8.999999E+09,8.999999E+09,8.999999E+09,8.999999E+09,8.999999E+09]];
	LOCAL CONST Robtarget Tr_meulage_bavure_P536 :=[[196.97015625,69.9323125,20],[0.556756906187995,-0.499958359592072,-0.443222724632126,0.493575731226376],[0,0,0,0],[8.999999E+09,8.999999E+09,8.999999E+09,8.999999E+09,8.999999E+09,8.999999E+09]];
	LOCAL CONST Robtarget Tr_meulage_bavure_P537 :=[[198.0001875,73.207125,20],[0.557085260907631,-0.501199738480464,-0.442874750513149,0.49225683294852],[0,0,0,0],[8.999999E+09,8.999999E+09,8.999999E+09,8.999999E+09,8.999999E+09,8.999999E+09]];
	LOCAL CONST Robtarget Tr_meulage_bavure_P538 :=[[198.21478125,74.337953125,20],[0.556715316771657,-0.501846645291047,-0.443233137569013,0.491693386616786],[0,0,0,0],[8.999999E+09,8.999999E+09,8.999999E+09,8.999999E+09,8.999999E+09,8.999999E+09]];
	LOCAL CONST Robtarget Tr_meulage_bavure_P539 :=[[198.242375,76.4633515625,20],[0.555505015360066,-0.501767707629148,-0.444447730629304,0.492046298867154],[0,0,0,0],[8.999999E+09,8.999999E+09,8.999999E+09,8.999999E+09,8.999999E+09,8.999999E+09]];
	LOCAL CONST Robtarget Tr_meulage_bavure_P540 :=[[198.171265625,77.5245703125,20],[0.553433020900331,-0.50090529482097,-0.446538551253499,0.493365077039181],[0,0,0,0],[8.999999E+09,8.999999E+09,8.999999E+09,8.999999E+09,8.999999E+09,8.999999E+09]];
	LOCAL CONST Robtarget Tr_meulage_bavure_P541 :=[[198.1095625,79.0714453125,20],[0.55057880174278,-0.499338006314779,-0.44941395413436,0.4955316703808],[0,0,0,0],[8.999999E+09,8.999999E+09,8.999999E+09,8.999999E+09,8.999999E+09,8.999999E+09]];
	LOCAL CONST Robtarget Tr_meulage_bavure_P542 :=[[197.898984375,86.595671875,20],[0.547088289921776,-0.497215811090394,-0.452911078584196,0.498339638327003],[0,0,0,0],[8.999999E+09,8.999999E+09,8.999999E+09,8.999999E+09,8.999999E+09,8.999999E+09]];
	LOCAL CONST Robtarget Tr_meulage_bavure_P543 :=[[197.927671875,87.3577578125,20],[0.543186633965197,-0.494723608781873,-0.456790153085258,0.501537224580336],[0,0,0,0],[8.999999E+09,8.999999E+09,8.999999E+09,8.999999E+09,8.999999E+09,8.999999E+09]];
	LOCAL CONST Robtarget Tr_meulage_bavure_P544 :=[[197.9638125,95.10409375,20],[0.539114729453636,-0.49207574044707,-0.460803635092097,0.504853230192212],[0,0,0,0],[8.999999E+09,8.999999E+09,8.999999E+09,8.999999E+09,8.999999E+09,8.999999E+09]];
	LOCAL CONST Robtarget Tr_meulage_bavure_P545 :=[[197.887515625,97.1987578125,20],[0.535076872863968,-0.489454351950437,-0.464749847695087,0.508069637500893],[0,0,0,0],[8.999999E+09,8.999999E+09,8.999999E+09,8.999999E+09,8.999999E+09,8.999999E+09]];
	LOCAL CONST Robtarget Tr_meulage_bavure_P546 :=[[197.87921875,100.32959375,20],[0.531226870759147,-0.486994978687208,-0.468484132065601,0.511034754708162],[0,0,0,0],[8.999999E+09,8.999999E+09,8.999999E+09,8.999999E+09,8.999999E+09,8.999999E+09]];
	LOCAL CONST Robtarget Tr_meulage_bavure_P547 :=[[197.930234375,101.4933203125,20],[0.527690498555941,-0.484808744791088,-0.471893984273727,0.513633416274817],[0,0,0,0],[8.999999E+09,8.999999E+09,8.999999E+09,8.999999E+09,8.999999E+09,8.999999E+09]];
	LOCAL CONST Robtarget Tr_meulage_bavure_P548 :=[[197.88396875,104.7469140625,20],[0.524518361829746,-0.482955774566138,-0.474941643013406,0.515814543851167],[0,0,0,0],[8.999999E+09,8.999999E+09,8.999999E+09,8.999999E+09,8.999999E+09,8.999999E+09]];
	LOCAL CONST Robtarget Tr_meulage_bavure_P549 :=[[197.5910625,110.33715625,20],[0.521722448994115,-0.481436317591407,-0.477623761741003,0.517590862110202],[0,0,0,0],[8.999999E+09,8.999999E+09,8.999999E+09,8.999999E+09,8.999999E+09,8.999999E+09]];
	LOCAL CONST Robtarget Tr_meulage_bavure_P550 :=[[197.583984375,110.7712734375,20],[0.519286803794282,-0.480251866844645,-0.479963187570008,0.518974660629004],[0,0,0,0],[8.999999E+09,8.999999E+09,8.999999E+09,8.999999E+09,8.999999E+09,8.999999E+09]];
	LOCAL CONST Robtarget Tr_meulage_bavure_P551 :=[[197.598203125,111.3843671875,20],[0.517213971528147,-0.479365203785704,-0.481959558521991,0.520013166184144],[0,0,0,0],[8.999999E+09,8.999999E+09,8.999999E+09,8.999999E+09,8.999999E+09,8.999999E+09]];
	LOCAL CONST Robtarget Tr_meulage_bavure_P552 :=[[197.476984375,114.2478046875,20],[0.51545266968024,-0.478777825030864,-0.483667500314139,0.520716898821327],[0,0,0,0],[8.999999E+09,8.999999E+09,8.999999E+09,8.999999E+09,8.999999E+09,8.999999E+09]];
	LOCAL CONST Robtarget Tr_meulage_bavure_P553 :=[[197.42553125,117.438875,20],[0.51400979722862,-0.478448921474584,-0.485078843934965,0.521132490888372],[0,0,0,0],[8.999999E+09,8.999999E+09,8.999999E+09,8.999999E+09,8.999999E+09,8.999999E+09]];
	LOCAL CONST Robtarget Tr_meulage_bavure_P554 :=[[197.37084375,118.19546875,20],[0.51285476284149,-0.478396688348523,-0.486226666920058,0.521248721038025],[0,0,0,0],[8.999999E+09,8.999999E+09,8.999999E+09,8.999999E+09,8.999999E+09,8.999999E+09]];
	LOCAL CONST Robtarget Tr_meulage_bavure_P555 :=[[197.434015625,119.891109375,20],[0.51198853780264,-0.478590078648298,-0.487107492447153,0.521100340222473],[0,0,0,0],[8.999999E+09,8.999999E+09,8.999999E+09,8.999999E+09,8.999999E+09,8.999999E+09]];
	LOCAL CONST Robtarget Tr_meulage_bavure_P556 :=[[197.423515625,120.578765625,20],[0.511397980911549,-0.479018780141731,-0.4877329308965,0.520701163346337],[0,0,0,0],[8.999999E+09,8.999999E+09,8.999999E+09,8.999999E+09,8.999999E+09,8.999999E+09]];
	LOCAL CONST Robtarget Tr_meulage_bavure_P557 :=[[197.39978125,121.2391640625,20],[0.511059362749325,-0.479686532874659,-0.488125682042463,0.520050455682449],[0,0,0,0],[8.999999E+09,8.999999E+09,8.999999E+09,8.999999E+09,8.999999E+09,8.999999E+09]];
	LOCAL CONST Robtarget Tr_meulage_bavure_P558 :=[[197.249390625,126.4974375,20],[0.510961920094526,-0.480560325266301,-0.488291958486508,0.519182678130417],[0,0,0,0],[8.999999E+09,8.999999E+09,8.999999E+09,8.999999E+09,8.999999E+09,8.999999E+09]];
	LOCAL CONST Robtarget Tr_meulage_bavure_P559 :=[[197.2373125,128.434265625,20],[0.511064233327587,-0.481599174153241,-0.488267892752313,0.518140955508651],[0,0,0,0],[8.999999E+09,8.999999E+09,8.999999E+09,8.999999E+09,8.999999E+09,8.999999E+09]];
	LOCAL CONST Robtarget Tr_meulage_bavure_P560 :=[[196.931453125,133.64740625,20],[0.51133503200629,-0.482762333959704,-0.488079809441906,0.51696722678334],[0,0,0,0],[8.999999E+09,8.999999E+09,8.999999E+09,8.999999E+09,8.999999E+09,8.999999E+09]];
	LOCAL CONST Robtarget Tr_meulage_bavure_P561 :=[[196.9716875,135.947046875,20],[0.511702865924955,-0.484024197696998,-0.487795647322437,0.51568998390627],[0,0,0,0],[8.999999E+09,8.999999E+09,8.999999E+09,8.999999E+09,8.999999E+09,8.999999E+09]];
	LOCAL CONST Robtarget Tr_meulage_bavure_P562 :=[[196.946109375,137.87646875,20],[0.512121068155827,-0.485311225638352,-0.487456213387865,0.514384550555223],[0,0,0,0],[8.999999E+09,8.999999E+09,8.999999E+09,8.999999E+09,8.999999E+09,8.999999E+09]];
	LOCAL CONST Robtarget Tr_meulage_bavure_P563 :=[[196.85534375,142.292578125,20],[0.512537967184181,-0.486572236179579,-0.487109992444672,0.513104420595324],[0,0,0,0],[8.999999E+09,8.999999E+09,8.999999E+09,8.999999E+09,8.999999E+09,8.999999E+09]];
	LOCAL CONST Robtarget Tr_meulage_bavure_P564 :=[[196.852046875,143.471796875,20],[0.51291543550198,-0.487758720600421,-0.486793120533836,0.511900033505552],[0,0,0,0],[8.999999E+09,8.999999E+09,8.999999E+09,8.999999E+09,8.999999E+09,8.999999E+09]];
	LOCAL CONST Robtarget Tr_meulage_bavure_P565 :=[[196.95075,144.457765625,20],[0.513205262848461,-0.48885696402937,-0.486554226699572,0.510787834022514],[0,0,0,0],[8.999999E+09,8.999999E+09,8.999999E+09,8.999999E+09,8.999999E+09,8.999999E+09]];
	LOCAL CONST Robtarget Tr_meulage_bavure_P566 :=[[196.9685,145.540734375,20],[0.513398723392118,-0.489820081173679,-0.486401349769006,0.509815423306556],[0,0,0,0],[8.999999E+09,8.999999E+09,8.999999E+09,8.999999E+09,8.999999E+09,8.999999E+09]];
	LOCAL CONST Robtarget Tr_meulage_bavure_P567 :=[[197.20984375,149.507234375,20],[0.51346761349123,-0.490656010323682,-0.486364549795122,0.508976634170427],[0,0,0,0],[8.999999E+09,8.999999E+09,8.999999E+09,8.999999E+09,8.999999E+09,8.999999E+09]];
	LOCAL CONST Robtarget Tr_meulage_bavure_P568 :=[[197.236265625,151.1625625,20],[0.513414524389609,-0.491348278312041,-0.486441989980807,0.50828789669743],[0,0,0,0],[8.999999E+09,8.999999E+09,8.999999E+09,8.999999E+09,8.999999E+09,8.999999E+09]];
	LOCAL CONST Robtarget Tr_meulage_bavure_P569 :=[[197.339296875,155.87625,20],[0.513238739704485,-0.491877444173987,-0.486634987693797,0.507768613377861],[0,0,0,0],[8.999999E+09,8.999999E+09,8.999999E+09,8.999999E+09,8.999999E+09,8.999999E+09]];
	LOCAL CONST Robtarget Tr_meulage_bavure_P570 :=[[197.3044375,157.525453125,20],[0.512914743078441,-0.492236309094448,-0.486969870716183,0.507427066046457],[0,0,0,0],[8.999999E+09,8.999999E+09,8.999999E+09,8.999999E+09,8.999999E+09,8.999999E+09]];
	LOCAL CONST Robtarget Tr_meulage_bavure_P571 :=[[197.37096875,164.16390625,20],[0.512425258479691,-0.492397862473761,-0.487463839258688,0.507290552758942],[0,0,0,0],[8.999999E+09,8.999999E+09,8.999999E+09,8.999999E+09,8.999999E+09,8.999999E+09]];
	LOCAL CONST Robtarget Tr_meulage_bavure_P572 :=[[197.330390625,166.267125,20],[0.511736601980082,-0.492330059192087,-0.488149964511482,0.5073917373758],[0,0,0,0],[8.999999E+09,8.999999E+09,8.999999E+09,8.999999E+09,8.999999E+09,8.999999E+09]];
	LOCAL CONST Robtarget Tr_meulage_bavure_P573 :=[[197.466125,171.515046875,20],[0.510779934816662,-0.491987720817061,-0.489095404500801,0.507777142110708],[0,0,0,0],[8.999999E+09,8.999999E+09,8.999999E+09,8.999999E+09,8.999999E+09,8.999999E+09]];
	LOCAL CONST Robtarget Tr_meulage_bavure_P574 :=[[197.4815,172.705078125,20],[0.509498088035626,-0.491298022599363,-0.49035362501225,0.508518705374093],[0,0,0,0],[8.999999E+09,8.999999E+09,8.999999E+09,8.999999E+09,8.999999E+09,8.999999E+09]];
	LOCAL CONST Robtarget Tr_meulage_bavure_P575 :=[[197.499390625,173.644140625,20],[0.507808351283477,-0.490181654773505,-0.492001276385297,0.509693405613123],[0,0,0,0],[8.999999E+09,8.999999E+09,8.999999E+09,8.999999E+09,8.999999E+09,8.999999E+09]];
	LOCAL CONST Robtarget Tr_meulage_bavure_P576 :=[[197.362484375,180.21759375,20],[0.505625934889061,-0.488546377220477,-0.494113176088603,0.511387348775803],[0,0,0,0],[8.999999E+09,8.999999E+09,8.999999E+09,8.999999E+09,8.999999E+09,8.999999E+09]];
	LOCAL CONST Robtarget Tr_meulage_bavure_P577 :=[[197.411859375,183.889671875,20],[0.502864205089686,-0.486311108474903,-0.496761462998809,0.513670269621196],[0,0,0,0],[8.999999E+09,8.999999E+09,8.999999E+09,8.999999E+09,8.999999E+09,8.999999E+09]];
	LOCAL CONST Robtarget Tr_meulage_bavure_P578 :=[[197.560421875,190.301671875,20],[0.499446158233086,-0.483394201192286,-0.50000218963281,0.516605644222243],[0,0,0,0],[8.999999E+09,8.999999E+09,8.999999E+09,8.999999E+09,8.999999E+09,8.999999E+09]];
	LOCAL CONST Robtarget Tr_meulage_bavure_P579 :=[[197.567015625,193.150875,20],[0.495303653541238,-0.479722902520145,-0.503875177066297,0.520240361297311],[0,0,0,0],[8.999999E+09,8.999999E+09,8.999999E+09,8.999999E+09,8.999999E+09,8.999999E+09]];
	LOCAL CONST Robtarget Tr_meulage_bavure_P580 :=[[197.502265625,196.09615625,20],[0.490367478722645,-0.475258447270092,-0.508415538409049,0.524578673235821],[0,0,0,0],[8.999999E+09,8.999999E+09,8.999999E+09,8.999999E+09,8.999999E+09,8.999999E+09]];
	LOCAL CONST Robtarget Tr_meulage_bavure_P581 :=[[197.3591875,200.7161875,20],[0.484614181861629,-0.46998006498207,-0.513606994231731,0.529599555073717],[0,0,0,0],[8.999999E+09,8.999999E+09,8.999999E+09,8.999999E+09,8.999999E+09,8.999999E+09]];
	LOCAL CONST Robtarget Tr_meulage_bavure_P582 :=[[196.776921875,205.48446875,20],[0.478059800260105,-0.463871244543124,-0.519387737525647,0.535274391288498],[0,0,0,0],[8.999999E+09,8.999999E+09,8.999999E+09,8.999999E+09,8.999999E+09,8.999999E+09]];
	LOCAL CONST Robtarget Tr_meulage_bavure_P583 :=[[196.27496875,210.62515625,20],[0.470734193387022,-0.456961388461825,-0.52568365609022,0.541527748458868],[0,0,0,0],[8.999999E+09,8.999999E+09,8.999999E+09,8.999999E+09,8.999999E+09,8.999999E+09]];
	LOCAL CONST Robtarget Tr_meulage_bavure_P584 :=[[196.012578125,211.897578125,20],[0.462688555802663,-0.449339689769591,-0.532410102113877,0.548226802239826],[0,0,0,0],[8.999999E+09,8.999999E+09,8.999999E+09,8.999999E+09,8.999999E+09,8.999999E+09]];
	LOCAL CONST Robtarget Tr_meulage_bavure_P585 :=[[195.66296875,214.245421875,20],[0.45405142942733,-0.441089590179646,-0.539409666738207,0.555260735420331],[0,0,0,0],[8.999999E+09,8.999999E+09,8.999999E+09,8.999999E+09,8.999999E+09,8.999999E+09]];
	LOCAL CONST Robtarget Tr_meulage_bavure_P586 :=[[195.42828125,215.07525,20],[0.444936868191166,-0.432348862883482,-0.546560706148279,0.562474033696038],[0,0,0,0],[8.999999E+09,8.999999E+09,8.999999E+09,8.999999E+09,8.999999E+09,8.999999E+09]];
	LOCAL CONST Robtarget Tr_meulage_bavure_P587 :=[[195.215703125,215.848265625,20],[0.435509875435362,-0.423266134349026,-0.553707031951904,0.569724012727673],[0,0,0,0],[8.999999E+09,8.999999E+09,8.999999E+09,8.999999E+09,8.999999E+09,8.999999E+09]];
	LOCAL CONST Robtarget Tr_meulage_bavure_P588 :=[[194.34521875,219.92346875,20],[0.425935214128574,-0.414028740082265,-0.560721024982998,0.576846017489203],[0,0,0,0],[8.999999E+09,8.999999E+09,8.999999E+09,8.999999E+09,8.999999E+09,8.999999E+09]];
	LOCAL CONST Robtarget Tr_meulage_bavure_P589 :=[[193.6485625,222.21253125,20],[0.416386072269695,-0.404772116186006,-0.567467160248621,0.583749256802512],[0,0,0,0],[8.999999E+09,8.999999E+09,8.999999E+09,8.999999E+09,8.999999E+09,8.999999E+09]];
	LOCAL CONST Robtarget Tr_meulage_bavure_P590 :=[[192.216125,225.1095,20],[0.406991561966914,-0.395641690991649,-0.573872534666168,0.590335357905003],[0,0,0,0],[8.999999E+09,8.999999E+09,8.999999E+09,8.999999E+09,8.999999E+09,8.999999E+09]];
	LOCAL CONST Robtarget Tr_meulage_bavure_P591 :=[[191.526734375,227.15521875,20],[0.397849481304488,-0.386735059397334,-0.579890368489767,0.596555902318879],[0,0,0,0],[8.999999E+09,8.999999E+09,8.999999E+09,8.999999E+09,8.999999E+09,8.999999E+09]];
	LOCAL CONST Robtarget Tr_meulage_bavure_P592 :=[[191.05309375,228.159796875,20],[0.389007602167415,-0.378099368041788,-0.585511552296207,0.602403664887627],[0,0,0,0],[8.999999E+09,8.999999E+09,8.999999E+09,8.999999E+09,8.999999E+09,8.999999E+09]];
	LOCAL CONST Robtarget Tr_meulage_bavure_P593 :=[[189.55603125,230.654359375,20],[0.380449878439608,-0.369708837687875,-0.590762179409333,0.607925417062244],[0,0,0,0],[8.999999E+09,8.999999E+09,8.999999E+09,8.999999E+09,8.999999E+09,8.999999E+09]];
	LOCAL CONST Robtarget Tr_meulage_bavure_P594 :=[[188.223515625,233.596625,20],[0.372089457674067,-0.361514142047017,-0.595730600188835,0.613157412567506],[0,0,0,0],[8.999999E+09,8.999999E+09,8.999999E+09,8.999999E+09,8.999999E+09,8.999999E+09]];
	LOCAL CONST Robtarget Tr_meulage_bavure_P595 :=[[187.378421875,235.114078125,20],[0.363831870106622,-0.35339615800965,-0.600469960459271,0.6182017084939],[0,0,0,0],[8.999999E+09,8.999999E+09,8.999999E+09,8.999999E+09,8.999999E+09,8.999999E+09]];
	LOCAL CONST Robtarget Tr_meulage_bavure_P596 :=[[186.973578125,236.08740625,20],[0.355534291764644,-0.345230425462154,-0.605074694356317,0.623133962294018],[0,0,0,0],[8.999999E+09,8.999999E+09,8.999999E+09,8.999999E+09,8.999999E+09,8.999999E+09]];
	LOCAL CONST Robtarget Tr_meulage_bavure_P597 :=[[186.587640625,237.10253125,20],[0.3470563688248,-0.336888027327106,-0.609624915454501,0.62802531506213],[0,0,0,0],[8.999999E+09,8.999999E+09,8.999999E+09,8.999999E+09,8.999999E+09,8.999999E+09]];
	LOCAL CONST Robtarget Tr_meulage_bavure_P598 :=[[186.04296875,237.93903125,20],[0.338269725466571,-0.328228811861906,-0.614169435674174,0.632957616416897],[0,0,0,0],[8.999999E+09,8.999999E+09,8.999999E+09,8.999999E+09,8.999999E+09,8.999999E+09]];
	LOCAL CONST Robtarget Tr_meulage_bavure_P599 :=[[185.23725,239.375609375,20],[0.329075267665939,-0.319171448217623,-0.618753017507843,0.637952786793972],[0,0,0,0],[8.999999E+09,8.999999E+09,8.999999E+09,8.999999E+09,8.999999E+09,8.999999E+09]];
	LOCAL CONST Robtarget Tr_meulage_bavure_P600 :=[[182.822453125,243.005609375,20],[0.319419551997363,-0.309664824353545,-0.62338206025877,0.643019170248776],[0,0,0,0],[8.999999E+09,8.999999E+09,8.999999E+09,8.999999E+09,8.999999E+09,8.999999E+09]];
	LOCAL CONST Robtarget Tr_meulage_bavure_P601 :=[[179.732546875,247.647515625,20],[0.309323835127442,-0.299730067336048,-0.628023785449753,0.648125587109583],[0,0,0,0],[8.999999E+09,8.999999E+09,8.999999E+09,8.999999E+09,8.999999E+09,8.999999E+09]];
	LOCAL CONST Robtarget Tr_meulage_bavure_P602 :=[[179.003359375,248.5080625,20],[0.298855679007099,-0.28943300549982,-0.632625918075571,0.653221452672513],[0,0,0,0],[8.999999E+09,8.999999E+09,8.999999E+09,8.999999E+09,8.999999E+09,8.999999E+09]];
	LOCAL CONST Robtarget Tr_meulage_bavure_P603 :=[[176.3124375,250.900328125,20],[0.288108074197399,-0.278871493265929,-0.637137472844894,0.658240281753341],[0,0,0,0],[8.999999E+09,8.999999E+09,8.999999E+09,8.999999E+09,8.999999E+09,8.999999E+09]];
	LOCAL CONST Robtarget Tr_meulage_bavure_P604 :=[[175.4530625,251.849125,20],[0.277226620179513,-0.268191871112388,-0.641492683307744,0.663103052772125],[0,0,0,0],[8.999999E+09,8.999999E+09,8.999999E+09,8.999999E+09,8.999999E+09,8.999999E+09]];
	LOCAL CONST Robtarget Tr_meulage_bavure_P605 :=[[173.79303125,253.32525,20],[0.266348499075339,-0.257518954618794,-0.645627009628096,0.667763602999625],[0,0,0,0],[8.999999E+09,8.999999E+09,8.999999E+09,8.999999E+09,8.999999E+09,8.999999E+09]];
	LOCAL CONST Robtarget Tr_meulage_bavure_P606 :=[[172.833671875,254.371765625,20],[0.255579039481533,-0.246954579181905,-0.649504836164167,0.672187665907479],[0,0,0,0],[8.999999E+09,8.999999E+09,8.999999E+09,8.999999E+09,8.999999E+09,8.999999E+09]];
	LOCAL CONST Robtarget Tr_meulage_bavure_P607 :=[[171.835625,255.384453125,20],[0.24496020638397,-0.236558287517955,-0.653143697512287,0.676341618041411],[0,0,0,0],[8.999999E+09,8.999999E+09,8.999999E+09,8.999999E+09,8.999999E+09,8.999999E+09]];
	LOCAL CONST Robtarget Tr_meulage_bavure_P608 :=[[169.96515625,256.785953125,20],[0.234487916760538,-0.22630564464428,-0.656532129682311,0.680269604487992],[0,0,0,0],[8.999999E+09,8.999999E+09,8.999999E+09,8.999999E+09,8.999999E+09,8.999999E+09]];
	LOCAL CONST Robtarget Tr_meulage_bavure_P609 :=[[167.427734375,259.1613125,20],[0.224081782747706,-0.216131598022023,-0.659722045533385,0.683989261329667],[0,0,0,0],[8.999999E+09,8.999999E+09,8.999999E+09,8.999999E+09,8.999999E+09,8.999999E+09]];
	LOCAL CONST Robtarget Tr_meulage_bavure_P610 :=[[167.3435,259.22015625,20],[0.213629328151924,-0.205929848597438,-0.662757663271789,0.687537407989203],[0,0,0,0],[8.999999E+09,8.999999E+09,8.999999E+09,8.999999E+09,8.999999E+09,8.999999E+09]];
	LOCAL CONST Robtarget Tr_meulage_bavure_P611 :=[[166.99071875,259.50678125,20],[0.20300458902943,-0.195581832553998,-0.66568123014538,0.69094528252239],[0,0,0,0],[8.999999E+09,8.999999E+09,8.999999E+09,8.999999E+09,8.999999E+09,8.999999E+09]];
	LOCAL CONST Robtarget Tr_meulage_bavure_P612 :=[[164.57921875,261.1981875,20],[0.192115374236905,-0.184985599945552,-0.668491046864081,0.694256243081158],[0,0,0,0],[8.999999E+09,8.999999E+09,8.999999E+09,8.999999E+09,8.999999E+09,8.999999E+09]];
	LOCAL CONST Robtarget Tr_meulage_bavure_P613 :=[[164.3856875,261.31365625,20],[0.180911879482151,-0.174104074836585,-0.671206948177068,0.697452432576129],[0,0,0,0],[8.999999E+09,8.999999E+09,8.999999E+09,8.999999E+09,8.999999E+09,8.999999E+09]];
	LOCAL CONST Robtarget Tr_meulage_bavure_P614 :=[[159.45159375,264.3151875,20],[0.169410509493069,-0.162945360471106,-0.673797950555364,0.70053209105767],[0,0,0,0],[8.999999E+09,8.999999E+09,8.999999E+09,8.999999E+09,8.999999E+09,8.999999E+09]];
	LOCAL CONST Robtarget Tr_meulage_bavure_P615 :=[[156.9999375,265.75865625,20],[0.157707166912385,-0.151610868175561,-0.67624918509222,0.703441279580342],[0,0,0,0],[8.999999E+09,8.999999E+09,8.999999E+09,8.999999E+09,8.999999E+09,8.999999E+09]];
	LOCAL CONST Robtarget Tr_meulage_bavure_P616 :=[[156.77721875,265.869875,20],[0.145960642520499,-0.140249296974879,-0.678515280752183,0.706146329962029],[0,0,0,0],[8.999999E+09,8.999999E+09,8.999999E+09,8.999999E+09,8.999999E+09,8.999999E+09]];
	LOCAL CONST Robtarget Tr_meulage_bavure_P617 :=[[153.837828125,267.192375,20],[0.134369066972975,-0.129052170216997,-0.680565755350058,0.708604786780262],[0,0,0,0],[8.999999E+09,8.999999E+09,8.999999E+09,8.999999E+09,8.999999E+09,8.999999E+09]];
	LOCAL CONST Robtarget Tr_meulage_bavure_P618 :=[[151.61359375,268.03978125,20],[0.123153469724389,-0.118232447879033,-0.682380410875514,0.710782164954031],[0,0,0,0],[8.999999E+09,8.999999E+09,8.999999E+09,8.999999E+09,8.999999E+09,8.999999E+09]];
	LOCAL CONST Robtarget Tr_meulage_bavure_P619 :=[[150.777703125,268.32134375,20],[0.112538538223628,-0.108000255968493,-0.683934570404306,0.712674207145949],[0,0,0,0],[8.999999E+09,8.999999E+09,8.999999E+09,8.999999E+09,8.999999E+09,8.999999E+09]];
	LOCAL CONST Robtarget Tr_meulage_bavure_P620 :=[[147.324578125,269.26025,20],[0.102725392033291,-0.0985513447257392,-0.685243529313122,0.714266359153818],[0,0,0,0],[8.999999E+09,8.999999E+09,8.999999E+09,8.999999E+09,8.999999E+09,8.999999E+09]];
	LOCAL CONST Robtarget Tr_meulage_bavure_P621 :=[[144.201109375,270.2108125,20],[0.0938862495457982,-0.0900417819394286,-0.686294094636664,0.715596440263811],[0,0,0,0],[8.999999E+09,8.999999E+09,8.999999E+09,8.999999E+09,8.999999E+09,8.999999E+09]];
	LOCAL CONST Robtarget Tr_meulage_bavure_P622 :=[[139.504765625,271.383125,20],[0.0861608587617447,-0.0826118050359282,-0.687136070363109,0.716655856664891],[0,0,0,0],[8.999999E+09,8.999999E+09,8.999999E+09,8.999999E+09,8.999999E+09,8.999999E+09]];
	LOCAL CONST Robtarget Tr_meulage_bavure_P623 :=[[137.05090625,272.1169375,20],[0.0796689217420805,-0.0763714049032936,-0.687782215556839,0.71747884664656],[0,0,0,0],[8.999999E+09,8.999999E+09,8.999999E+09,8.999999E+09,8.999999E+09,8.999999E+09]];
	LOCAL CONST Robtarget Tr_meulage_bavure_P624 :=[[136.521171875,272.21625,20],[0.0745182676432689,-0.0714230297156304,-0.688258308530526,0.718085147703519],[0,0,0,0],[8.999999E+09,8.999999E+09,8.999999E+09,8.999999E+09,8.999999E+09,8.999999E+09]];
	LOCAL CONST Robtarget Tr_meulage_bavure_P625 :=[[134.061765625,272.86078125,20],[0.0707808315219947,-0.0678306389736018,-0.688567166423668,0.718515369097119],[0,0,0,0],[8.999999E+09,8.999999E+09,8.999999E+09,8.999999E+09,8.999999E+09,8.999999E+09]];
	LOCAL CONST Robtarget Tr_meulage_bavure_P626 :=[[133.05609375,273.01178125,20],[0.0685138145589592,-0.0656559708967384,-0.688766106896634,0.718746409167129],[0,0,0,0],[8.999999E+09,8.999999E+09,8.999999E+09,8.999999E+09,8.999999E+09,8.999999E+09]];
	LOCAL CONST Robtarget Tr_meulage_bavure_P627 :=[[129.749875,273.06775,20],[0.067760017222189,-0.0649318951864941,-0.68882514439665,0.718827065086223],[0,0,0,0],[8.999999E+09,8.999999E+09,8.999999E+09,8.999999E+09,8.999999E+09,8.999999E+09]];
	LOCAL CONST Robtarget Tr_meulage_bavure_degg1 :=[[131.616867145896,282.882677411363,19.5739246113115],[0.067760017222189,-0.0649318951864941,-0.68882514439665,0.718827065086223],[0,0,0,0],[8.999999E+09,8.999999E+09,8.999999E+09,8.999999E+09,8.999999E+09,8.999999E+09]];
	LOCAL CONST Robtarget Tr_meulage_bavure_degg2 :=[[167.089717917915,469.366298227253,11.4784922262304],[0.067760017222189,-0.0649318951864941,-0.68882514439665,0.718827065086223],[0,0,0,0],[8.999999E+09,8.999999E+09,8.999999E+09,8.999999E+09,8.999999E+09,8.999999E+09]];
	LOCAL PROC Tr_pick()
		!!Programme Tr_pick - 04/04/2023 09:18:53;
		 CONST Robtarget Ppick :=[[-93.6973796577624,-28.893648402371,42.3720274076437],[0.00726739553894396,0.752949986585257,-0.657983845213,0.00841202128240375],[0,0,0,0],[8.999999E+09,8.999999E+09,8.999999E+09,8.999999E+09,8.999999E+09,8.999999E+09]];
		 VAR Pose Ref :=[[0,0,0],[1,0,0,0]];
		LocalisationPieceTable 105 \model:=0;
		MoveJ Reltool(Ppick,0,0,-200),V1000,Z0,Tool_Prehenseur \Wobj:=Wobj_vision;
		MoveL Reltool(Ppick,0,0,-100),V500,Z0,Tool_Prehenseur \Wobj:=Wobj_vision;
		MoveL Reltool(Ppick,0,0,-10),V200,Z0,Tool_Prehenseur \Wobj:=Wobj_vision;
		MoveL Ppick,V100,Fine,Tool_Prehenseur \Wobj:=Wobj_vision;
		Gripper_Close;
		MoveL Reltool(Ppick,0,0,-200),V500,Z0,Tool_Prehenseur \Wobj:=Wobj_vision;
		LocalisationPiecePrehenseur 105 \model:=0,Ref;
	ENDPROC
	LOCAL PROC Tr_Cut()
		!!Programme Tr_Cut - 04/04/2023 09:18:53;
		confJ \off;
		confL \off;
		Tool := ToolOffset(Tool_M2_D490_S180);
		MoveAbsJ [[0,-40,40,0,90,0],[8.999999E+09,8.999999E+09,8.999999E+09,8.999999E+09,8.999999E+09,8.999999E+09]] ,V1000,Z0,Tool_M2_D490_S180 \Wobj:=Wobj_Part_0;
		Movej Reltool(Coupe_0,-200,0,-45.2220625),V1000,Z0,Tool_M2_D490_S180 \Wobj:=Wobj_Part_0;
		MoveL Reltool(Coupe_0,0,0,-45.2220625),V500,Z0,Tool_M2_D490_S180 \Wobj:=Wobj_Part_0;
		MoveL Reltool(Coupe_0,0,0,-35.2220625),vitesse_Tronconnage,Z0,Tool_M2_D490_S180 \Wobj:=Wobj_Part_0;
		MoveL Coupe_0,vitesse_Tronconnage,Fine,Tool_M2_D490_S180 \Wobj:=Wobj_Part_0;
		MoveL Reltool(Coupe_0,0,0,35.2220625),vitesse_Tronconnage,Z0,Tool_M2_D490_S180 \Wobj:=Wobj_Part_0;
		MoveL Reltool(Coupe_0,-200,0,35.2220625),V500,Z0,Tool_M2_D490_S180 \Wobj:=Wobj_Part_0;
	ENDPROC
	LOCAL PROC Tr_meulage_motif_1()
		!!Programme Tr_meulage_motif_1 - 04/04/2023 09:18:53;
		 CONST Speeddata vitesse_Meulage :=[50, 500, 0, 0];
		confJ \off;
		confL \off;
		Tool := ToolOffset(Tool_M1_D500_S0);
		MoveAbsJ [[0,-40,40,0,90,0],[8.999999E+09,8.999999E+09,8.999999E+09,8.999999E+09,8.999999E+09,8.999999E+09]] ,V1000,Z0,Tool_M1_D500_S0 \Wobj:=Wobj_Part_0;
		MoveJ Tr_meulage_motif_1_App1,V2000,Z100,Tool,\Wobj:=Wobj_Part_0;
		MoveJ Tr_meulage_motif_1_App2,V500,Z0,Tool,\Wobj:=Wobj_Part_0;
		MoveL Tr_meulage_motif_1_P0,[12.5,500,0,0],z0,Tool \wobj:=Wobj_Part_0;
		MoveL Tr_meulage_motif_1_P1,[12.5,500,0,0],z0,Tool \wobj:=Wobj_Part_0;
		MoveL Tr_meulage_motif_1_P2,[12.5,500,0,0],z0,Tool \wobj:=Wobj_Part_0;
		MoveL Tr_meulage_motif_1_P3,[12.5,500,0,0],z0,Tool \wobj:=Wobj_Part_0;
		MoveL Tr_meulage_motif_1_P4,[12.5,500,0,0],z0,Tool \wobj:=Wobj_Part_0;
		MoveL Tr_meulage_motif_1_P5,[12.5,500,0,0],z0,Tool \wobj:=Wobj_Part_0;
		MoveL Tr_meulage_motif_1_P6,[12.5,500,0,0],z0,Tool \wobj:=Wobj_Part_0;
		MoveL Tr_meulage_motif_1_P7,[12.5,500,0,0],z0,Tool \wobj:=Wobj_Part_0;
		MoveL Tr_meulage_motif_1_P8,[12.5,500,0,0],z0,Tool \wobj:=Wobj_Part_0;
		MoveL Tr_meulage_motif_1_P9,[12.5,500,0,0],z0,Tool \wobj:=Wobj_Part_0;
		MoveL Tr_meulage_motif_1_P10,[12.5,500,0,0],z0,Tool \wobj:=Wobj_Part_0;
		MoveL Tr_meulage_motif_1_P11,[12.5,500,0,0],z0,Tool \wobj:=Wobj_Part_0;
		MoveL Tr_meulage_motif_1_P12,[12.5,500,0,0],z0,Tool \wobj:=Wobj_Part_0;
		MoveL Tr_meulage_motif_1_P13,[12.5,500,0,0],z0,Tool \wobj:=Wobj_Part_0;
		MoveL Tr_meulage_motif_1_P14,[12.5,500,0,0],z0,Tool \wobj:=Wobj_Part_0;
		MoveL Tr_meulage_motif_1_P15,[12.5,500,0,0],z0,Tool \wobj:=Wobj_Part_0;
		MoveL Tr_meulage_motif_1_P16,[12.5,500,0,0],z0,Tool \wobj:=Wobj_Part_0;
		MoveL Tr_meulage_motif_1_P17,[12.5,500,0,0],z0,Tool \wobj:=Wobj_Part_0;
		MoveL Tr_meulage_motif_1_P18,[12.5,500,0,0],z0,Tool \wobj:=Wobj_Part_0;
		MoveL Tr_meulage_motif_1_P19,[12.5,500,0,0],z0,Tool \wobj:=Wobj_Part_0;
		MoveL Tr_meulage_motif_1_P20,[12.5,500,0,0],z0,Tool \wobj:=Wobj_Part_0;
		MoveL Tr_meulage_motif_1_P21,[12.5,500,0,0],z0,Tool \wobj:=Wobj_Part_0;
		MoveL Tr_meulage_motif_1_P22,[12.5,500,0,0],z0,Tool \wobj:=Wobj_Part_0;
		MoveL Tr_meulage_motif_1_P23,[12.5,500,0,0],z0,Tool \wobj:=Wobj_Part_0;
		MoveL Tr_meulage_motif_1_P24,[12.5,500,0,0],z0,Tool \wobj:=Wobj_Part_0;
		MoveL Tr_meulage_motif_1_P25,[12.5,500,0,0],z0,Tool \wobj:=Wobj_Part_0;
		MoveL Tr_meulage_motif_1_P26,[12.5,500,0,0],z0,Tool \wobj:=Wobj_Part_0;
		MoveL Tr_meulage_motif_1_P27,[12.5,500,0,0],z0,Tool \wobj:=Wobj_Part_0;
		MoveL Tr_meulage_motif_1_P28,[12.5,500,0,0],z0,Tool \wobj:=Wobj_Part_0;
		MoveL Tr_meulage_motif_1_P29,[12.5,500,0,0],z0,Tool \wobj:=Wobj_Part_0;
		MoveL Tr_meulage_motif_1_P30,[12.5,500,0,0],z0,Tool \wobj:=Wobj_Part_0;
		MoveL Tr_meulage_motif_1_P31,[12.5,500,0,0],z0,Tool \wobj:=Wobj_Part_0;
		MoveL Tr_meulage_motif_1_P32,[12.5,500,0,0],z0,Tool \wobj:=Wobj_Part_0;
		MoveL Tr_meulage_motif_1_P33,[12.5,500,0,0],z0,Tool \wobj:=Wobj_Part_0;
		MoveL Tr_meulage_motif_1_P34,[12.5,500,0,0],z0,Tool \wobj:=Wobj_Part_0;
		MoveL Tr_meulage_motif_1_P35,[12.5,500,0,0],z0,Tool \wobj:=Wobj_Part_0;
		MoveL Tr_meulage_motif_1_P36,[12.5,500,0,0],z0,Tool \wobj:=Wobj_Part_0;
		MoveL Tr_meulage_motif_1_P37,[12.5,500,0,0],z0,Tool \wobj:=Wobj_Part_0;
		MoveL Tr_meulage_motif_1_P38,[12.5,500,0,0],z0,Tool \wobj:=Wobj_Part_0;
		MoveL Tr_meulage_motif_1_P39,[12.5,500,0,0],z0,Tool \wobj:=Wobj_Part_0;
		MoveL Tr_meulage_motif_1_P40,[12.5,500,0,0],z0,Tool \wobj:=Wobj_Part_0;
		MoveL Tr_meulage_motif_1_P41,[12.5,500,0,0],z0,Tool \wobj:=Wobj_Part_0;
		MoveL Tr_meulage_motif_1_P42,[12.5,500,0,0],z0,Tool \wobj:=Wobj_Part_0;
		MoveL Tr_meulage_motif_1_P43,[12.5,500,0,0],z0,Tool \wobj:=Wobj_Part_0;
		MoveL Tr_meulage_motif_1_P44,[12.5,500,0,0],z0,Tool \wobj:=Wobj_Part_0;
		MoveL Tr_meulage_motif_1_P45,[12.5,500,0,0],z0,Tool \wobj:=Wobj_Part_0;
		MoveL Tr_meulage_motif_1_P46,[12.5,500,0,0],z0,Tool \wobj:=Wobj_Part_0;
		MoveL Tr_meulage_motif_1_P47,[12.5,500,0,0],z0,Tool \wobj:=Wobj_Part_0;
		MoveL Tr_meulage_motif_1_P48,[12.5,500,0,0],z0,Tool \wobj:=Wobj_Part_0;
		MoveL Tr_meulage_motif_1_P49,[12.5,500,0,0],z0,Tool \wobj:=Wobj_Part_0;
		MoveL Tr_meulage_motif_1_P50,[12.5,500,0,0],z0,Tool \wobj:=Wobj_Part_0;
		MoveL Tr_meulage_motif_1_P51,[12.5,500,0,0],z0,Tool \wobj:=Wobj_Part_0;
		MoveL Tr_meulage_motif_1_P52,[12.5,500,0,0],z0,Tool \wobj:=Wobj_Part_0;
		MoveL Tr_meulage_motif_1_P53,[12.5,500,0,0],z0,Tool \wobj:=Wobj_Part_0;
		MoveL Tr_meulage_motif_1_P54,[12.5,500,0,0],z0,Tool \wobj:=Wobj_Part_0;
		MoveL Tr_meulage_motif_1_P55,[12.5,500,0,0],z0,Tool \wobj:=Wobj_Part_0;
		MoveL Tr_meulage_motif_1_P56,[12.5,500,0,0],z0,Tool \wobj:=Wobj_Part_0;
		MoveL Tr_meulage_motif_1_P57,[12.5,500,0,0],z0,Tool \wobj:=Wobj_Part_0;
		MoveL Tr_meulage_motif_1_P58,[12.5,500,0,0],z0,Tool \wobj:=Wobj_Part_0;
		MoveL Tr_meulage_motif_1_P59,[12.5,500,0,0],z0,Tool \wobj:=Wobj_Part_0;
		MoveL Tr_meulage_motif_1_P60,[12.5,500,0,0],z0,Tool \wobj:=Wobj_Part_0;
		MoveL Tr_meulage_motif_1_P61,[12.5,500,0,0],z0,Tool \wobj:=Wobj_Part_0;
		MoveL Tr_meulage_motif_1_P62,[12.5,500,0,0],z0,Tool \wobj:=Wobj_Part_0;
		MoveL Tr_meulage_motif_1_P63,[12.5,500,0,0],z0,Tool \wobj:=Wobj_Part_0;
		MoveL Tr_meulage_motif_1_P64,[12.5,500,0,0],z0,Tool \wobj:=Wobj_Part_0;
		MoveL Tr_meulage_motif_1_P65,[12.5,500,0,0],z0,Tool \wobj:=Wobj_Part_0;
		MoveL Tr_meulage_motif_1_P66,[12.5,500,0,0],z0,Tool \wobj:=Wobj_Part_0;
		MoveL Tr_meulage_motif_1_P67,[12.5,500,0,0],z0,Tool \wobj:=Wobj_Part_0;
		MoveL Tr_meulage_motif_1_P68,[12.5,500,0,0],z0,Tool \wobj:=Wobj_Part_0;
		MoveL Tr_meulage_motif_1_P69,[12.5,500,0,0],z0,Tool \wobj:=Wobj_Part_0;
		MoveL Tr_meulage_motif_1_P70,[12.5,500,0,0],z0,Tool \wobj:=Wobj_Part_0;
		MoveL Tr_meulage_motif_1_P71,[12.5,500,0,0],z0,Tool \wobj:=Wobj_Part_0;
		MoveL Tr_meulage_motif_1_P72,[12.5,500,0,0],z0,Tool \wobj:=Wobj_Part_0;
		MoveL Tr_meulage_motif_1_P73,[12.5,500,0,0],z0,Tool \wobj:=Wobj_Part_0;
		MoveL Tr_meulage_motif_1_P74,[12.5,500,0,0],z0,Tool \wobj:=Wobj_Part_0;
		MoveL Tr_meulage_motif_1_P75,[12.5,500,0,0],z0,Tool \wobj:=Wobj_Part_0;
		MoveL Tr_meulage_motif_1_P76,[12.5,500,0,0],z0,Tool \wobj:=Wobj_Part_0;
		MoveL Tr_meulage_motif_1_P77,[12.5,500,0,0],z0,Tool \wobj:=Wobj_Part_0;
		MoveL Tr_meulage_motif_1_P78,[12.5,500,0,0],z0,Tool \wobj:=Wobj_Part_0;
		MoveL Tr_meulage_motif_1_P79,[12.5,500,0,0],z0,Tool \wobj:=Wobj_Part_0;
		MoveL Tr_meulage_motif_1_P80,[12.5,500,0,0],z0,Tool \wobj:=Wobj_Part_0;
		MoveL Tr_meulage_motif_1_P81,[12.5,500,0,0],z0,Tool \wobj:=Wobj_Part_0;
		MoveL Tr_meulage_motif_1_P82,[12.5,500,0,0],z0,Tool \wobj:=Wobj_Part_0;
		MoveL Tr_meulage_motif_1_P83,[12.5,500,0,0],z0,Tool \wobj:=Wobj_Part_0;
		MoveL Tr_meulage_motif_1_P84,[12.5,500,0,0],z0,Tool \wobj:=Wobj_Part_0;
		MoveL Tr_meulage_motif_1_P85,[12.5,500,0,0],z0,Tool \wobj:=Wobj_Part_0;
		MoveL Tr_meulage_motif_1_P86,[12.5,500,0,0],z0,Tool \wobj:=Wobj_Part_0;
		MoveL Tr_meulage_motif_1_P87,[12.5,500,0,0],z0,Tool \wobj:=Wobj_Part_0;
		MoveL Tr_meulage_motif_1_P88,[12.5,500,0,0],z0,Tool \wobj:=Wobj_Part_0;
		MoveL Tr_meulage_motif_1_P89,[12.5,500,0,0],z0,Tool \wobj:=Wobj_Part_0;
		MoveL Tr_meulage_motif_1_P90,[12.5,500,0,0],z0,Tool \wobj:=Wobj_Part_0;
		MoveL Tr_meulage_motif_1_P91,[12.5,500,0,0],z0,Tool \wobj:=Wobj_Part_0;
		MoveL Tr_meulage_motif_1_P92,[12.5,500,0,0],z0,Tool \wobj:=Wobj_Part_0;
		MoveL Tr_meulage_motif_1_P93,[12.5,500,0,0],z0,Tool \wobj:=Wobj_Part_0;
		MoveL Tr_meulage_motif_1_P94,[12.5,500,0,0],z0,Tool \wobj:=Wobj_Part_0;
		MoveL Tr_meulage_motif_1_P95,[12.5,500,0,0],z0,Tool \wobj:=Wobj_Part_0;
		MoveL Tr_meulage_motif_1_P96,[12.5,500,0,0],z0,Tool \wobj:=Wobj_Part_0;
		MoveL Tr_meulage_motif_1_P97,[12.5,500,0,0],z0,Tool \wobj:=Wobj_Part_0;
		MoveL Tr_meulage_motif_1_P98,[12.5,500,0,0],z0,Tool \wobj:=Wobj_Part_0;
		MoveL Tr_meulage_motif_1_P99,[12.5,500,0,0],z0,Tool \wobj:=Wobj_Part_0;
		MoveL Tr_meulage_motif_1_P100,[12.5,500,0,0],z0,Tool \wobj:=Wobj_Part_0;
		MoveL Tr_meulage_motif_1_P101,[12.5,500,0,0],z0,Tool \wobj:=Wobj_Part_0;
		MoveL Tr_meulage_motif_1_P102,[12.5,500,0,0],z0,Tool \wobj:=Wobj_Part_0;
		MoveL Tr_meulage_motif_1_P103,[12.5,500,0,0],z0,Tool \wobj:=Wobj_Part_0;
		MoveL Tr_meulage_motif_1_P104,[12.5,500,0,0],z0,Tool \wobj:=Wobj_Part_0;
		MoveL Tr_meulage_motif_1_P105,[12.5,500,0,0],z0,Tool \wobj:=Wobj_Part_0;
		MoveL Tr_meulage_motif_1_P106,[12.5,500,0,0],z0,Tool \wobj:=Wobj_Part_0;
		MoveL Tr_meulage_motif_1_P107,[12.5,500,0,0],z0,Tool \wobj:=Wobj_Part_0;
